LIN {X 0,Y 389.049,Z 504.507,A -85,B 0,C 180,E1 -11720.074,E2 -11720.074} C_VEL
LIN {X 0,Y 389.166,Z 500.329,A -85,B 0,C 180,E1 -11723.41,E2 -11723.41} C_VEL
LIN {X 0,Y 389.351,Z 496.924,A -85,B 0,C 180,E1 -11726.247,E2 -11726.247} C_VEL
LIN {X 0,Y 389.873,Z 499.181,A -85,B 0,C 180,E1 -11727.366,E2 -11727.366} C_VEL
LIN {X 0,Y 389.734,Z 506.684,A -85,B 0,C 180,E1 -11730.926,E2 -11730.926} C_VEL
LIN {X 0,Y 389.566,Z 513.106,A -85,B 0,C 180,E1 -11734.005,E2 -11734.005} C_VEL
LIN {X 0,Y 389.452,Z 518.341,A -85,B 0,C 180,E1 -11736.549,E2 -11736.549} C_VEL
LIN {X 0,Y 389.235,Z 525.161,A -85,B 0,C 180,E1 -11739.865,E2 -11739.865} C_VEL
LIN {X 0,Y 389.197,Z 528.183,A -85,B 0,C 180,E1 -11741.336,E2 -11741.336} C_VEL
LIN {X 0,Y 391.433,Z 539.991,A -85,B 0,C 180,E1 -11741.917,E2 -11741.917} C_VEL
LIN {X 0,Y 392.651,Z 549.622,A -85,B 0,C 180,E1 -11742.527,E2 -11742.527} C_VEL
LIN {X 0,Y 392.07,Z 559.282,A -85,B 0,C 180,E1 -11743.262,E2 -11743.262} C_VEL
LIN {X 0,Y 391.528,Z 567.985,A -85,B 0,C 180,E1 -11744.109,E2 -11744.109} C_VEL
LIN {X 0,Y 391.008,Z 575.053,A -85,B 0,C 180,E1 -11744.949,E2 -11744.949} C_VEL
LIN {X 0,Y 390.507,Z 581.055,A -85,B 0,C 180,E1 -11745.798,E2 -11745.798} C_VEL
LIN {X 0,Y 390.083,Z 586.933,A -85,B 0,C 180,E1 -11746.793,E2 -11746.793} C_VEL
LIN {X 0,Y 389.589,Z 593.354,A -85,B 0,C 180,E1 -11748.128,E2 -11748.128} C_VEL
LIN {X 0,Y 389.178,Z 599.487,A -85,B 0,C 180,E1 -11749.789,E2 -11749.789} C_VEL
LIN {X 0,Y 388.96,Z 602.788,A -85,B 0,C 180,E1 -11750.983,E2 -11750.983} C_VEL
LIN {X 0,Y 388.792,Z 605.13,A -85,B 0,C 180,E1 -11752.076,E2 -11752.076} C_VEL
LIN {X 0,Y 388.611,Z 607.077,A -85,B 0,C 180,E1 -11753.358,E2 -11753.358} C_VEL
LIN {X 0,Y 388.533,Z 608.221,A -85,B 0,C 180,E1 -11754.631,E2 -11754.631} C_VEL
LIN {X 0,Y 388.489,Z 608.513,A -85,B 0,C 180,E1 -11756.322,E2 -11756.322} C_VEL
LIN {X 0,Y 388.489,Z 608.255,A -85,B 0,C 180,E1 -11757.131,E2 -11757.131} C_VEL
LIN {X 0,Y 388.571,Z 607.186,A -85,B 0,C 180,E1 -11758.364,E2 -11758.364} C_VEL
LIN {X 0,Y 388.745,Z 605.399,A -85,B 0,C 180,E1 -11759.588,E2 -11759.588} C_VEL
LIN {X 0,Y 388.944,Z 601.354,A -85,B 0,C 180,E1 -11761.39,E2 -11761.39} C_VEL
LIN {X 0,Y 389.209,Z 597.195,A -85,B 0,C 180,E1 -11762.713,E2 -11762.713} C_VEL
LIN {X 0,Y 389.481,Z 593.091,A -85,B 0,C 180,E1 -11763.762,E2 -11763.762} C_VEL
LIN {X 0,Y 389.868,Z 587.471,A -85,B 0,C 180,E1 -11764.936,E2 -11764.936} C_VEL
LIN {X 0,Y 390.201,Z 582.47,A -85,B 0,C 180,E1 -11765.81,E2 -11765.81} C_VEL
LIN {X 0,Y 390.697,Z 575.482,A -85,B 0,C 180,E1 -11766.827,E2 -11766.827} C_VEL
LIN {X 0,Y 391.169,Z 568.265,A -85,B 0,C 180,E1 -11767.694,E2 -11767.694} C_VEL
LIN {X 0,Y 391.642,Z 559.908,A -85,B 0,C 180,E1 -11768.515,E2 -11768.515} C_VEL
LIN {X 0,Y 392.198,Z 550.305,A -85,B 0,C 180,E1 -11769.262,E2 -11769.262} C_VEL
LIN {X 0,Y 391.067,Z 540.77,A -85,B 0,C 180,E1 -11769.873,E2 -11769.873} C_VEL
LIN {X 0,Y 389.276,Z 529.916,A -85,B 0,C 180,E1 -11770.385,E2 -11770.385} C_VEL
LIN {X 0,Y 388.993,Z 528.206,A -85,B 0,C 180,E1 -11770.473,E2 -11770.473} C_VEL
LIN {X 0,Y 389.132,Z 520.919,A -85,B 0,C 180,E1 -11774.281,E2 -11774.281} C_VEL
LIN {X 0,Y 389.368,Z 513.777,A -85,B 0,C 180,E1 -11778.019,E2 -11778.019} C_VEL
LIN {X 0,Y 389.503,Z 506.789,A -85,B 0,C 180,E1 -11781.7,E2 -11781.7} C_VEL
LIN {X 0,Y 389.702,Z 499.725,A -85,B 0,C 180,E1 -11785.345,E2 -11785.345} C_VEL
LIN {X 0,Y 389.768,Z 496.75,A -85,B 0,C 180,E1 -11786.899,E2 -11786.899} C_VEL
LIN {X 0,Y 390.538,Z 496.652,A -85,B 0,C 180,E1 -11789.999,E2 -11789.999} C_VEL
LIN {X 0,Y 390.316,Z 496.677,A -85,B 0,C 180,E1 -11793.096,E2 -11793.096} C_VEL
LIN {X 0,Y 390.332,Z 496.678,A -85,B 0,C 180,E1 -11796.201,E2 -11796.201} C_VEL
LIN {X 0,Y 390.316,Z 496.68,A -85,B 0,C 180,E1 -11798.282,E2 -11798.282} C_VEL
LIN {X 0,Y 390.171,Z 496.698,A -85,B 0,C 180,E1 -11802.483,E2 -11802.483} C_VEL
LIN {X 0,Y 390.129,Z 496.7,A -85,B 0,C 180,E1 -11804.935,E2 -11804.935} C_VEL
LIN {X 0,Y 389.455,Z 496.787,A -85,B 0,C 180,E1 -11805.797,E2 -11805.797} C_VEL
LIN {X 0,Y 386.606,Z 497.139,A -85,B 0,C 180,E1 -11807.198,E2 -11807.198} C_VEL
LIN {X 0,Y 384.191,Z 497.444,A -85,B 0,C 180,E1 -11808.33,E2 -11808.33} C_VEL
LIN {X 0,Y 383.141,Z 497.57,A -85,B 0,C 180,E1 -11809.206,E2 -11809.206} C_VEL
LIN {X 0,Y 383.048,Z 497.581,A -85,B 0,C 180,E1 -11809.502,E2 -11809.502} C_VEL
LIN {X 0,Y 383.038,Z 497.583,A -85,B 0,C 180,E1 -11813.45,E2 -11813.45} C_VEL
LIN {X 0,Y 383.079,Z 497.582,A -85,B 0,C 180,E1 -11816.123,E2 -11816.123} C_VEL
LIN {X 0,Y 383.049,Z 497.585,A -85,B 0,C 180,E1 -11818.491,E2 -11818.491} C_VEL
LIN {X 0,Y 383.011,Z 497.591,A -85,B 0,C 180,E1 -11822.149,E2 -11822.149} C_VEL
LIN {X 0,Y 383.017,Z 497.587,A -85,B 0,C 180,E1 -11824.667,E2 -11824.667} C_VEL
LIN {X 0,Y 383.001,Z 497.591,A -85,B 0,C 180,E1 -11827.904,E2 -11827.904} C_VEL
LIN {X 0,Y 382.984,Z 497.59,A -85,B 0,C 180,E1 -11831.347,E2 -11831.347} C_VEL
LIN {X 0,Y 383.009,Z 497.59,A -85,B 0,C 180,E1 -11834.305,E2 -11834.305} C_VEL
LIN {X 0,Y 383.073,Z 497.578,A -85,B 0,C 180,E1 -11837.249,E2 -11837.249} C_VEL
LIN {X 0,Y 383.02,Z 497.588,A -85,B 0,C 180,E1 -11840.412,E2 -11840.412} C_VEL
LIN {X 0,Y 383.024,Z 497.589,A -85,B 0,C 180,E1 -11844.044,E2 -11844.044} C_VEL
LIN {X 0,Y 382.984,Z 497.592,A -85,B 0,C 180,E1 -11847.578,E2 -11847.578} C_VEL
LIN {X 0,Y 382.989,Z 497.592,A -85,B 0,C 180,E1 -11850.3,E2 -11850.3} C_VEL
LIN {X 0,Y 383.078,Z 497.582,A -85,B 0,C 180,E1 -11854.02,E2 -11854.02} C_VEL
LIN {X 0,Y 383.006,Z 497.588,A -85,B 0,C 180,E1 -11857.335,E2 -11857.335} C_VEL
LIN {X 0,Y 383.058,Z 497.58,A -85,B 0,C 180,E1 -11860.716,E2 -11860.716} C_VEL
LIN {X 0,Y 383.079,Z 497.582,A -85,B 0,C 180,E1 -11864.026,E2 -11864.026} C_VEL
LIN {X 0,Y 383.139,Z 497.571,A -85,B 0,C 180,E1 -11867.284,E2 -11867.284} C_VEL
LIN {X 0,Y 383.154,Z 497.569,A -85,B 0,C 180,E1 -11870.498,E2 -11870.498} C_VEL
LIN {X 0,Y 383.27,Z 497.554,A -85,B 0,C 180,E1 -11872.625,E2 -11872.625} C_VEL
LIN {X 0,Y 383.197,Z 497.563,A -85,B 0,C 180,E1 -11874.738,E2 -11874.738} C_VEL
LIN {X 0,Y 383.386,Z 497.544,A -85,B 0,C 180,E1 -11877.899,E2 -11877.899} C_VEL
LIN {X 0,Y 383.517,Z 497.527,A -85,B 0,C 180,E1 -11880,E2 -11880} C_VEL
LIN {X 0,Y 383.251,Z 497.558,A -85,B 0,C 180,E1 -11883.154,E2 -11883.154} C_VEL
LIN {X 0,Y 383.285,Z 497.553,A -85,B 0,C 180,E1 -11886.316,E2 -11886.316} C_VEL
LIN {X 0,Y 383.258,Z 497.556,A -85,B 0,C 180,E1 -11888.436,E2 -11888.436} C_VEL
LIN {X 0,Y 383.096,Z 497.58,A -85,B 0,C 180,E1 -11891.642,E2 -11891.642} C_VEL
LIN {X 0,Y 383.107,Z 497.575,A -85,B 0,C 180,E1 -11894.882,E2 -11894.882} C_VEL
LIN {X 0,Y 383.06,Z 497.581,A -85,B 0,C 180,E1 -11898.174,E2 -11898.174} C_VEL
LIN {X 0,Y 382.99,Z 497.593,A -85,B 0,C 180,E1 -11901.531,E2 -11901.531} C_VEL
LIN {X 0,Y 383.049,Z 497.582,A -85,B 0,C 180,E1 -11904.96,E2 -11904.96} C_VEL
LIN {X 0,Y 383.046,Z 497.582,A -85,B 0,C 180,E1 -11908.492,E2 -11908.492} C_VEL
LIN {X 0,Y 383.005,Z 497.587,A -85,B 0,C 180,E1 -11912.427,E2 -11912.427} C_VEL
LIN {X 0,Y 383.024,Z 497.587,A -85,B 0,C 180,E1 -11915.956,E2 -11915.956} C_VEL
LIN {X 0,Y 383.013,Z 497.59,A -85,B 0,C 180,E1 -11919.587,E2 -11919.587} C_VEL
LIN {X 0,Y 383.002,Z 497.588,A -85,B 0,C 180,E1 -11922.779,E2 -11922.779} C_VEL
LIN {X 0,Y 382.996,Z 497.592,A -85,B 0,C 180,E1 -11925.79,E2 -11925.79} C_VEL
LIN {X 0,Y 383.013,Z 497.587,A -85,B 0,C 180,E1 -11928.792,E2 -11928.792} C_VEL
LIN {X 0,Y 383.002,Z 497.59,A -85,B 0,C 180,E1 -11932.096,E2 -11932.096} C_VEL
LIN {X 0,Y 383.051,Z 497.676,A -85,B 0,C 180,E1 -11933.309,E2 -11933.309} C_VEL
LIN {X 0,Y 384.076,Z 503.252,A -85,B 0,C 180,E1 -11936.103,E2 -11936.103} C_VEL
LIN {X 0,Y 384.649,Z 507.173,A -85,B 0,C 180,E1 -11938.004,E2 -11938.004} C_VEL
LIN {X 0,Y 384.181,Z 513.651,A -85,B 0,C 180,E1 -11940.982,E2 -11940.982} C_VEL
LIN {X 0,Y 383.461,Z 521.478,A -85,B 0,C 180,E1 -11944.488,E2 -11944.488} C_VEL
LIN {X 0,Y 382.882,Z 529.232,A -85,B 0,C 180,E1 -11947.897,E2 -11947.897} C_VEL
LIN {X 0,Y 382.364,Z 538.246,A -85,B 0,C 180,E1 -11951.793,E2 -11951.793} C_VEL
LIN {X 0,Y 382.008,Z 546.977,A -85,B 0,C 180,E1 -11955.524,E2 -11955.524} C_VEL
LIN {X 0,Y 383.204,Z 558.101,A -85,B 0,C 180,E1 -11955.964,E2 -11955.964} C_VEL
LIN {X 0,Y 384.171,Z 569.277,A -85,B 0,C 180,E1 -11956.589,E2 -11956.589} C_VEL
LIN {X 0,Y 384.332,Z 577.789,A -85,B 0,C 180,E1 -11957.216,E2 -11957.216} C_VEL
LIN {X 0,Y 383.755,Z 587.394,A -85,B 0,C 180,E1 -11958.111,E2 -11958.111} C_VEL
LIN {X 0,Y 383.292,Z 595.307,A -85,B 0,C 180,E1 -11959.034,E2 -11959.034} C_VEL
LIN {X 0,Y 382.818,Z 601.82,A -85,B 0,C 180,E1 -11959.956,E2 -11959.956} C_VEL
LIN {X 0,Y 382.428,Z 607.997,A -85,B 0,C 180,E1 -11961.014,E2 -11961.014} C_VEL
LIN {X 0,Y 382.075,Z 614.282,A -85,B 0,C 180,E1 -11962.337,E2 -11962.337} C_VEL
LIN {X 0,Y 381.784,Z 619.534,A -85,B 0,C 180,E1 -11963.745,E2 -11963.745} C_VEL
LIN {X 0,Y 381.734,Z 623.67,A -85,B 0,C 180,E1 -11965.248,E2 -11965.248} C_VEL
LIN {X 0,Y 381.61,Z 626.719,A -85,B 0,C 180,E1 -11966.833,E2 -11966.833} C_VEL
LIN {X 0,Y 381.628,Z 628.092,A -85,B 0,C 180,E1 -11967.89,E2 -11967.89} C_VEL
LIN {X 0,Y 381.669,Z 628.965,A -85,B 0,C 180,E1 -11968.945,E2 -11968.945} C_VEL
LIN {X 0,Y 381.681,Z 629.274,A -85,B 0,C 180,E1 -11970.001,E2 -11970.001} C_VEL
LIN {X 0,Y 381.669,Z 629.017,A -85,B 0,C 180,E1 -11971.056,E2 -11971.056} C_VEL
LIN {X 0,Y 381.623,Z 628.273,A -85,B 0,C 180,E1 -11972.111,E2 -11972.111} C_VEL
LIN {X 0,Y 381.599,Z 627.035,A -85,B 0,C 180,E1 -11973.168,E2 -11973.168} C_VEL
LIN {X 0,Y 381.736,Z 624.119,A -85,B 0,C 180,E1 -11974.753,E2 -11974.753} C_VEL
LIN {X 0,Y 381.751,Z 621.238,A -85,B 0,C 180,E1 -11975.884,E2 -11975.884} C_VEL
LIN {X 0,Y 382.042,Z 616.321,A -85,B 0,C 180,E1 -11977.399,E2 -11977.399} C_VEL
LIN {X 0,Y 382.397,Z 611.016,A -85,B 0,C 180,E1 -11978.722,E2 -11978.722} C_VEL
LIN {X 0,Y 382.939,Z 604.445,A -85,B 0,C 180,E1 -11980.041,E2 -11980.041} C_VEL
LIN {X 0,Y 383.679,Z 596.352,A -85,B 0,C 180,E1 -11981.357,E2 -11981.357} C_VEL
LIN {X 0,Y 384.433,Z 587.126,A -85,B 0,C 180,E1 -11982.539,E2 -11982.539} C_VEL
LIN {X 0,Y 385.246,Z 578.244,A -85,B 0,C 180,E1 -11983.451,E2 -11983.451} C_VEL
LIN {X 0,Y 385.214,Z 569.496,A -85,B 0,C 180,E1 -11984.227,E2 -11984.227} C_VEL
LIN {X 0,Y 384.556,Z 559.789,A -85,B 0,C 180,E1 -11984.96,E2 -11984.96} C_VEL
LIN {X 0,Y 382.593,Z 547.8,A -85,B 0,C 180,E1 -11985.73,E2 -11985.73} C_VEL
LIN {X 0,Y 382.063,Z 545.124,A -85,B 0,C 180,E1 -11985.881,E2 -11985.881} C_VEL
LIN {X 0,Y 382.441,Z 537.733,A -85,B 0,C 180,E1 -11989.317,E2 -11989.317} C_VEL
LIN {X 0,Y 382.895,Z 530.876,A -85,B 0,C 180,E1 -11992.672,E2 -11992.672} C_VEL
LIN {X 0,Y 383.459,Z 525.387,A -85,B 0,C 180,E1 -11995.513,E2 -11995.513} C_VEL
LIN {X 0,Y 384.131,Z 519.884,A -85,B 0,C 180,E1 -11998.574,E2 -11998.574} C_VEL
LIN {X 0,Y 384.904,Z 514.395,A -85,B 0,C 180,E1 -12001.973,E2 -12001.973} C_VEL
LIN {X 0,Y 385.185,Z 510.943,A -85,B 0,C 180,E1 -12004.446,E2 -12004.446} C_VEL
LIN {X 0,Y 384.805,Z 507.931,A -85,B 0,C 180,E1 -12007.064,E2 -12007.064} C_VEL
LIN {X 0,Y 384.399,Z 505.368,A -85,B 0,C 180,E1 -12009.835,E2 -12009.835} C_VEL
LIN {X 0,Y 384.03,Z 503.279,A -85,B 0,C 180,E1 -12012.944,E2 -12012.944} C_VEL
LIN {X 0,Y 383.811,Z 502.03,A -85,B 0,C 180,E1 -12015.907,E2 -12015.907} C_VEL
LIN {X 0,Y 383.693,Z 501.503,A -85,B 0,C 180,E1 -12018.746,E2 -12018.746} C_VEL
LIN {X 0,Y 383.687,Z 501.616,A -85,B 0,C 180,E1 -12021.966,E2 -12021.966} C_VEL
LIN {X 0,Y 383.733,Z 502.06,A -85,B 0,C 180,E1 -12024.121,E2 -12024.121} C_VEL
LIN {X 0,Y 383.785,Z 503.255,A -85,B 0,C 180,E1 -12027.392,E2 -12027.392} C_VEL
LIN {X 0,Y 383.465,Z 504.845,A -85,B 0,C 180,E1 -12030.34,E2 -12030.34} C_VEL
LIN {X 0,Y 383.059,Z 507.299,A -85,B 0,C 180,E1 -12034.029,E2 -12034.029} C_VEL
LIN {X 0,Y 382.756,Z 509.832,A -85,B 0,C 180,E1 -12037.32,E2 -12037.32} C_VEL
LIN {X 0,Y 382.535,Z 512.699,A -85,B 0,C 180,E1 -12040.689,E2 -12040.689} C_VEL
LIN {X 0,Y 382.316,Z 516.009,A -85,B 0,C 180,E1 -12044.276,E2 -12044.276} C_VEL
LIN {X 0,Y 385.469,Z 526.823,A -85,B 0,C 180,E1 -12045.088,E2 -12045.088} C_VEL
LIN {X 0,Y 386.98,Z 535.241,A -85,B 0,C 180,E1 -12045.792,E2 -12045.792} C_VEL
LIN {X 0,Y 386.311,Z 544.52,A -85,B 0,C 180,E1 -12046.588,E2 -12046.588} C_VEL
LIN {X 0,Y 385.581,Z 553.105,A -85,B 0,C 180,E1 -12047.5,E2 -12047.5} C_VEL
LIN {X 0,Y 384.783,Z 562.092,A -85,B 0,C 180,E1 -12048.677,E2 -12048.677} C_VEL
LIN {X 0,Y 383.992,Z 569.911,A -85,B 0,C 180,E1 -12049.987,E2 -12049.987} C_VEL
LIN {X 0,Y 383.385,Z 576.206,A -85,B 0,C 180,E1 -12051.302,E2 -12051.302} C_VEL
LIN {X 0,Y 382.925,Z 581.247,A -85,B 0,C 180,E1 -12052.619,E2 -12052.619} C_VEL
LIN {X 0,Y 382.358,Z 585.933,A -85,B 0,C 180,E1 -12054.198,E2 -12054.198} C_VEL
LIN {X 0,Y 382.23,Z 589.116,A -85,B 0,C 180,E1 -12055.782,E2 -12055.782} C_VEL
LIN {X 0,Y 381.996,Z 590.639,A -85,B 0,C 180,E1 -12056.836,E2 -12056.836} C_VEL
LIN {X 0,Y 381.838,Z 591.561,A -85,B 0,C 180,E1 -12057.89,E2 -12057.89} C_VEL
LIN {X 0,Y 381.72,Z 591.956,A -85,B 0,C 180,E1 -12058.945,E2 -12058.945} C_VEL
LIN {X 0,Y 381.684,Z 591.867,A -85,B 0,C 180,E1 -12060,E2 -12060} C_VEL
LIN {X 0,Y 381.708,Z 591.289,A -85,B 0,C 180,E1 -12061.055,E2 -12061.055} C_VEL
LIN {X 0,Y 381.79,Z 590.191,A -85,B 0,C 180,E1 -12062.11,E2 -12062.11} C_VEL
LIN {X 0,Y 381.823,Z 587.432,A -85,B 0,C 180,E1 -12063.694,E2 -12063.694} C_VEL
LIN {X 0,Y 381.942,Z 584.941,A -85,B 0,C 180,E1 -12064.75,E2 -12064.75} C_VEL
LIN {X 0,Y 382.161,Z 579.878,A -85,B 0,C 180,E1 -12066.335,E2 -12066.335} C_VEL
LIN {X 0,Y 382.451,Z 575.661,A -85,B 0,C 180,E1 -12067.391,E2 -12067.391} C_VEL
LIN {X 0,Y 382.636,Z 570.597,A -85,B 0,C 180,E1 -12068.45,E2 -12068.45} C_VEL
LIN {X 0,Y 383.015,Z 564.521,A -85,B 0,C 180,E1 -12069.506,E2 -12069.506} C_VEL
LIN {X 0,Y 383.538,Z 556.171,A -85,B 0,C 180,E1 -12070.692,E2 -12070.692} C_VEL
LIN {X 0,Y 384.064,Z 547.02,A -85,B 0,C 180,E1 -12071.746,E2 -12071.746} C_VEL
LIN {X 0,Y 384.611,Z 536.714,A -85,B 0,C 180,E1 -12072.667,E2 -12072.667} C_VEL
LIN {X 0,Y 384.733,Z 530.686,A -85,B 0,C 180,E1 -12073.117,E2 -12073.117} C_VEL
LIN {X 0,Y 382.871,Z 519.137,A -85,B 0,C 180,E1 -12073.823,E2 -12073.823} C_VEL
LIN {X 0,Y 381.887,Z 512.68,A -85,B 0,C 180,E1 -12074.148,E2 -12074.148} C_VEL
LIN {X 0,Y 381.92,Z 508.837,A -85,B 0,C 180,E1 -12077.123,E2 -12077.123} C_VEL
LIN {X 0,Y 381.983,Z 504.619,A -85,B 0,C 180,E1 -12080.461,E2 -12080.461} C_VEL
LIN {X 0,Y 382.102,Z 500.414,A -85,B 0,C 180,E1 -12083.869,E2 -12083.869} C_VEL
LIN {X 0,Y 382.27,Z 497.752,A -85,B 0,C 180,E1 -12086.112,E2 -12086.112} C_VEL
LIN {X 0,Y 382.862,Z 500.164,A -85,B 0,C 180,E1 -12087.317,E2 -12087.317} C_VEL
LIN {X 0,Y 382.73,Z 506.454,A -85,B 0,C 180,E1 -12090.338,E2 -12090.338} C_VEL
LIN {X 0,Y 382.597,Z 512.872,A -85,B 0,C 180,E1 -12093.441,E2 -12093.441} C_VEL
LIN {X 0,Y 382.4,Z 519.478,A -85,B 0,C 180,E1 -12096.677,E2 -12096.677} C_VEL
LIN {X 0,Y 382.185,Z 526.372,A -85,B 0,C 180,E1 -12100.062,E2 -12100.062} C_VEL
LIN {X 0,Y 382.151,Z 528.35,A -85,B 0,C 180,E1 -12101.037,E2 -12101.037} C_VEL
LIN {X 0,Y 384.343,Z 539.751,A -85,B 0,C 180,E1 -12101.606,E2 -12101.606} C_VEL
LIN {X 0,Y 385.754,Z 550.364,A -85,B 0,C 180,E1 -12102.296,E2 -12102.296} C_VEL
LIN {X 0,Y 385.116,Z 560.662,A -85,B 0,C 180,E1 -12103.116,E2 -12103.116} C_VEL
LIN {X 0,Y 384.561,Z 569.215,A -85,B 0,C 180,E1 -12103.985,E2 -12103.985} C_VEL
LIN {X 0,Y 383.934,Z 576.895,A -85,B 0,C 180,E1 -12104.944,E2 -12104.944} C_VEL
LIN {X 0,Y 383.288,Z 584.991,A -85,B 0,C 180,E1 -12106.196,E2 -12106.196} C_VEL
LIN {X 0,Y 382.687,Z 591.911,A -85,B 0,C 180,E1 -12107.582,E2 -12107.582} C_VEL
LIN {X 0,Y 382.305,Z 597.184,A -85,B 0,C 180,E1 -12108.913,E2 -12108.913} C_VEL
LIN {X 0,Y 382.055,Z 600.427,A -85,B 0,C 180,E1 -12109.921,E2 -12109.921} C_VEL
LIN {X 0,Y 381.823,Z 603.802,A -85,B 0,C 180,E1 -12111.257,E2 -12111.257} C_VEL
LIN {X 0,Y 381.653,Z 606.232,A -85,B 0,C 180,E1 -12112.577,E2 -12112.577} C_VEL
LIN {X 0,Y 381.468,Z 608.058,A -85,B 0,C 180,E1 -12114.158,E2 -12114.158} C_VEL
LIN {X 0,Y 381.394,Z 608.789,A -85,B 0,C 180,E1 -12116.019,E2 -12116.019} C_VEL
LIN {X 0,Y 381.443,Z 607.778,A -85,B 0,C 180,E1 -12117.945,E2 -12117.945} C_VEL
LIN {X 0,Y 381.561,Z 606.623,A -85,B 0,C 180,E1 -12118.953,E2 -12118.953} C_VEL
LIN {X 0,Y 381.692,Z 604.535,A -85,B 0,C 180,E1 -12120.188,E2 -12120.188} C_VEL
LIN {X 0,Y 381.985,Z 599.971,A -85,B 0,C 180,E1 -12122.023,E2 -12122.023} C_VEL
LIN {X 0,Y 382.355,Z 594.798,A -85,B 0,C 180,E1 -12123.529,E2 -12123.529} C_VEL
LIN {X 0,Y 382.779,Z 589.025,A -85,B 0,C 180,E1 -12124.816,E2 -12124.816} C_VEL
LIN {X 0,Y 383.162,Z 583.003,A -85,B 0,C 180,E1 -12125.913,E2 -12125.913} C_VEL
LIN {X 0,Y 383.69,Z 576.046,A -85,B 0,C 180,E1 -12126.953,E2 -12126.953} C_VEL
LIN {X 0,Y 384.168,Z 568.93,A -85,B 0,C 180,E1 -12127.832,E2 -12127.832} C_VEL
LIN {X 0,Y 384.594,Z 561.818,A -85,B 0,C 180,E1 -12128.563,E2 -12128.563} C_VEL
LIN {X 0,Y 385.161,Z 553.061,A -85,B 0,C 180,E1 -12129.289,E2 -12129.289} C_VEL
LIN {X 0,Y 385.144,Z 548.708,A -85,B 0,C 180,E1 -12129.608,E2 -12129.608} C_VEL
LIN {X 0,Y 383.53,Z 537.804,A -85,B 0,C 180,E1 -12130.272,E2 -12130.272} C_VEL
LIN {X 0,Y 381.934,Z 528.331,A -85,B 0,C 180,E1 -12130.726,E2 -12130.726} C_VEL
LIN {X 0,Y 382.066,Z 521.137,A -85,B 0,C 180,E1 -12134.53,E2 -12134.53} C_VEL
LIN {X 0,Y 382.332,Z 513.945,A -85,B 0,C 180,E1 -12138.334,E2 -12138.334} C_VEL
LIN {X 0,Y 382.444,Z 507.836,A -85,B 0,C 180,E1 -12141.546,E2 -12141.546} C_VEL
LIN {X 0,Y 382.671,Z 500.777,A -85,B 0,C 180,E1 -12145.259,E2 -12145.259} C_VEL
LIN {X 0,Y 382.743,Z 497.625,A -85,B 0,C 180,E1 -12146.973,E2 -12146.973} C_VEL
LIN {X 0,Y 383.485,Z 497.53,A -85,B 0,C 180,E1 -12149.999,E2 -12149.999} C_VEL
LIN {X 0,Y 383.252,Z 497.556,A -85,B 0,C 180,E1 -12153.153,E2 -12153.153} C_VEL
LIN {X 0,Y 383.289,Z 497.556,A -85,B 0,C 180,E1 -12156.316,E2 -12156.316} C_VEL
LIN {X 0,Y 383.261,Z 497.559,A -85,B 0,C 180,E1 -12158.435,E2 -12158.435} C_VEL
LIN {X 0,Y 383.098,Z 497.577,A -85,B 0,C 180,E1 -12161.642,E2 -12161.642} C_VEL
LIN {X 0,Y 383.108,Z 497.574,A -85,B 0,C 180,E1 -12164.921,E2 -12164.921} C_VEL
LIN {X 0,Y 383.09,Z 497.581,A -85,B 0,C 180,E1 -12168.172,E2 -12168.172} C_VEL
LIN {X 0,Y 383.048,Z 497.581,A -85,B 0,C 180,E1 -12169.502,E2 -12169.502} C_VEL
LIN {X 0,Y 382.358,Z 497.672,A -85,B 0,C 180,E1 -12170.379,E2 -12170.379} C_VEL
LIN {X 0,Y 379.491,Z 498.026,A -85,B 0,C 180,E1 -12171.805,E2 -12171.805} C_VEL
LIN {X 0,Y 377.085,Z 498.325,A -85,B 0,C 180,E1 -12172.957,E2 -12172.957} C_VEL
LIN {X 0,Y 376.067,Z 498.454,A -85,B 0,C 180,E1 -12173.848,E2 -12173.848} C_VEL
LIN {X 0,Y 375.99,Z 498.464,A -85,B 0,C 180,E1 -12174.15,E2 -12174.15} C_VEL
LIN {X 0,Y 376.019,Z 498.459,A -85,B 0,C 180,E1 -12176.651,E2 -12176.651} C_VEL
LIN {X 0,Y 375.976,Z 498.462,A -85,B 0,C 180,E1 -12179.078,E2 -12179.078} C_VEL
LIN {X 0,Y 375.951,Z 498.466,A -85,B 0,C 180,E1 -12182.828,E2 -12182.828} C_VEL
LIN {X 0,Y 375.957,Z 498.465,A -85,B 0,C 180,E1 -12185.415,E2 -12185.415} C_VEL
LIN {X 0,Y 375.975,Z 498.467,A -85,B 0,C 180,E1 -12188.27,E2 -12188.27} C_VEL
LIN {X 0,Y 375.934,Z 498.469,A -85,B 0,C 180,E1 -12191.6,E2 -12191.6} C_VEL
LIN {X 0,Y 375.98,Z 498.462,A -85,B 0,C 180,E1 -12195.26,E2 -12195.26} C_VEL
LIN {X 0,Y 375.988,Z 498.464,A -85,B 0,C 180,E1 -12198.389,E2 -12198.389} C_VEL
LIN {X 0,Y 375.966,Z 498.468,A -85,B 0,C 180,E1 -12201.912,E2 -12201.912} C_VEL
LIN {X 0,Y 375.977,Z 498.463,A -85,B 0,C 180,E1 -12205.332,E2 -12205.332} C_VEL
LIN {X 0,Y 375.955,Z 498.467,A -85,B 0,C 180,E1 -12208.438,E2 -12208.438} C_VEL
LIN {X 0,Y 375.981,Z 498.466,A -85,B 0,C 180,E1 -12212.14,E2 -12212.14} C_VEL
LIN {X 0,Y 376.004,Z 498.46,A -85,B 0,C 180,E1 -12214.539,E2 -12214.539} C_VEL
LIN {X 0,Y 375.961,Z 498.468,A -85,B 0,C 180,E1 -12218.045,E2 -12218.045} C_VEL
LIN {X 0,Y 376.021,Z 498.459,A -85,B 0,C 180,E1 -12221.474,E2 -12221.474} C_VEL
LIN {X 0,Y 376.057,Z 498.452,A -85,B 0,C 180,E1 -12224.832,E2 -12224.832} C_VEL
LIN {X 0,Y 376.056,Z 498.456,A -85,B 0,C 180,E1 -12228.137,E2 -12228.137} C_VEL
LIN {X 0,Y 376.255,Z 498.433,A -85,B 0,C 180,E1 -12231.877,E2 -12231.877} C_VEL
LIN {X 0,Y 376.17,Z 498.438,A -85,B 0,C 180,E1 -12234.64,E2 -12234.64} C_VEL
LIN {X 0,Y 376.352,Z 498.42,A -85,B 0,C 180,E1 -12237.86,E2 -12237.86} C_VEL
LIN {X 0,Y 376.486,Z 498.403,A -85,B 0,C 180,E1 -12240,E2 -12240} C_VEL
LIN {X 0,Y 376.189,Z 498.437,A -85,B 0,C 180,E1 -12243.213,E2 -12243.213} C_VEL
LIN {X 0,Y 376.244,Z 498.429,A -85,B 0,C 180,E1 -12246.435,E2 -12246.435} C_VEL
LIN {X 0,Y 376.203,Z 498.434,A -85,B 0,C 180,E1 -12248.595,E2 -12248.595} C_VEL
LIN {X 0,Y 376.048,Z 498.458,A -85,B 0,C 180,E1 -12251.863,E2 -12251.863} C_VEL
LIN {X 0,Y 376.055,Z 498.454,A -85,B 0,C 180,E1 -12255.167,E2 -12255.167} C_VEL
LIN {X 0,Y 376.006,Z 498.458,A -85,B 0,C 180,E1 -12258.527,E2 -12258.527} C_VEL
LIN {X 0,Y 375.96,Z 498.468,A -85,B 0,C 180,E1 -12261.954,E2 -12261.954} C_VEL
LIN {X 0,Y 376.004,Z 498.464,A -85,B 0,C 180,E1 -12265.461,E2 -12265.461} C_VEL
LIN {X 0,Y 375.974,Z 498.464,A -85,B 0,C 180,E1 -12269.079,E2 -12269.079} C_VEL
LIN {X 0,Y 375.955,Z 498.465,A -85,B 0,C 180,E1 -12272.828,E2 -12272.828} C_VEL
LIN {X 0,Y 375.955,Z 498.469,A -85,B 0,C 180,E1 -12275.416,E2 -12275.416} C_VEL
LIN {X 0,Y 375.973,Z 498.463,A -85,B 0,C 180,E1 -12278.271,E2 -12278.271} C_VEL
LIN {X 0,Y 375.932,Z 498.472,A -85,B 0,C 180,E1 -12281.601,E2 -12281.601} C_VEL
LIN {X 0,Y 375.951,Z 498.469,A -85,B 0,C 180,E1 -12285.265,E2 -12285.265} C_VEL
LIN {X 0,Y 375.979,Z 498.465,A -85,B 0,C 180,E1 -12289.139,E2 -12289.139} C_VEL
LIN {X 0,Y 376.03,Z 498.59,A -85,B 0,C 180,E1 -12293.185,E2 -12293.185} C_VEL
LIN {X 0,Y 377.019,Z 504.098,A -85,B 0,C 180,E1 -12295.998,E2 -12295.998} C_VEL
LIN {X 0,Y 377.631,Z 508.075,A -85,B 0,C 180,E1 -12297.968,E2 -12297.968} C_VEL
LIN {X 0,Y 377.085,Z 514.89,A -85,B 0,C 180,E1 -12301.16,E2 -12301.16} C_VEL
LIN {X 0,Y 376.359,Z 522.349,A -85,B 0,C 180,E1 -12304.565,E2 -12304.565} C_VEL
LIN {X 0,Y 375.767,Z 530.072,A -85,B 0,C 180,E1 -12308.034,E2 -12308.034} C_VEL
LIN {X 0,Y 375.253,Z 539.055,A -85,B 0,C 180,E1 -12312,E2 -12312} C_VEL
LIN {X 0,Y 374.905,Z 546.542,A -85,B 0,C 180,E1 -12315.272,E2 -12315.272} C_VEL
LIN {X 0,Y 375.987,Z 556.294,A -85,B 0,C 180,E1 -12315.644,E2 -12315.644} C_VEL
LIN {X 0,Y 376.795,Z 565.256,A -85,B 0,C 180,E1 -12316.121,E2 -12316.121} C_VEL
LIN {X 0,Y 377.407,Z 573.354,A -85,B 0,C 180,E1 -12316.677,E2 -12316.677} C_VEL
LIN {X 0,Y 377.212,Z 580.052,A -85,B 0,C 180,E1 -12317.218,E2 -12317.218} C_VEL
LIN {X 0,Y 376.716,Z 588.219,A -85,B 0,C 180,E1 -12318.022,E2 -12318.022} C_VEL
LIN {X 0,Y 376.215,Z 595.958,A -85,B 0,C 180,E1 -12318.962,E2 -12318.962} C_VEL
LIN {X 0,Y 375.683,Z 603.181,A -85,B 0,C 180,E1 -12320.036,E2 -12320.036} C_VEL
LIN {X 0,Y 375.223,Z 610.455,A -85,B 0,C 180,E1 -12321.383,E2 -12321.383} C_VEL
LIN {X 0,Y 374.979,Z 615.13,A -85,B 0,C 180,E1 -12322.462,E2 -12322.462} C_VEL
LIN {X 0,Y 374.677,Z 619.781,A -85,B 0,C 180,E1 -12323.797,E2 -12323.797} C_VEL
LIN {X 0,Y 374.645,Z 623.43,A -85,B 0,C 180,E1 -12325.158,E2 -12325.158} C_VEL
LIN {X 0,Y 374.522,Z 626.494,A -85,B 0,C 180,E1 -12326.773,E2 -12326.773} C_VEL
LIN {X 0,Y 374.526,Z 627.881,A -85,B 0,C 180,E1 -12327.85,E2 -12327.85} C_VEL
LIN {X 0,Y 374.569,Z 628.765,A -85,B 0,C 180,E1 -12328.925,E2 -12328.925} C_VEL
LIN {X 0,Y 374.612,Z 629.078,A -85,B 0,C 180,E1 -12330.001,E2 -12330.001} C_VEL
LIN {X 0,Y 374.569,Z 628.831,A -85,B 0,C 180,E1 -12331.076,E2 -12331.076} C_VEL
LIN {X 0,Y 374.521,Z 628.101,A -85,B 0,C 180,E1 -12332.151,E2 -12332.151} C_VEL
LIN {X 0,Y 374.512,Z 626.876,A -85,B 0,C 180,E1 -12333.228,E2 -12333.228} C_VEL
LIN {X 0,Y 374.648,Z 623.972,A -85,B 0,C 180,E1 -12334.843,E2 -12334.843} C_VEL
LIN {X 0,Y 374.76,Z 620.187,A -85,B 0,C 180,E1 -12336.318,E2 -12336.318} C_VEL
LIN {X 0,Y 375.111,Z 614.352,A -85,B 0,C 180,E1 -12338.078,E2 -12338.078} C_VEL
LIN {X 0,Y 375.575,Z 608.694,A -85,B 0,C 180,E1 -12339.424,E2 -12339.424} C_VEL
LIN {X 0,Y 376.253,Z 601.713,A -85,B 0,C 180,E1 -12340.766,E2 -12340.766} C_VEL
LIN {X 0,Y 377.146,Z 592.885,A -85,B 0,C 180,E1 -12342.102,E2 -12342.102} C_VEL
LIN {X 0,Y 377.795,Z 585.429,A -85,B 0,C 180,E1 -12343.036,E2 -12343.036} C_VEL
LIN {X 0,Y 378.525,Z 577.81,A -85,B 0,C 180,E1 -12343.831,E2 -12343.831} C_VEL
LIN {X 0,Y 378.406,Z 568.817,A -85,B 0,C 180,E1 -12344.652,E2 -12344.652} C_VEL
LIN {X 0,Y 377.711,Z 559.508,A -85,B 0,C 180,E1 -12345.376,E2 -12345.376} C_VEL
LIN {X 0,Y 375.376,Z 546.638,A -85,B 0,C 180,E1 -12346.25,E2 -12346.25} C_VEL
LIN {X 0,Y 375.047,Z 544.656,A -85,B 0,C 180,E1 -12346.378,E2 -12346.378} C_VEL
LIN {X 0,Y 375.536,Z 536.733,A -85,B 0,C 180,E1 -12350.186,E2 -12350.186} C_VEL
LIN {X 0,Y 376.189,Z 528.767,A -85,B 0,C 180,E1 -12354.269,E2 -12354.269} C_VEL
LIN {X 0,Y 376.902,Z 522.441,A -85,B 0,C 180,E1 -12357.786,E2 -12357.786} C_VEL
LIN {X 0,Y 377.729,Z 516.997,A -85,B 0,C 180,E1 -12361.144,E2 -12361.144} C_VEL
LIN {X 0,Y 378.164,Z 513.947,A -85,B 0,C 180,E1 -12363.248,E2 -12363.248} C_VEL
LIN {X 0,Y 378.176,Z 511.502,A -85,B 0,C 180,E1 -12365.177,E2 -12365.177} C_VEL
LIN {X 0,Y 377.657,Z 507.988,A -85,B 0,C 180,E1 -12368.593,E2 -12368.593} C_VEL
LIN {X 0,Y 377.209,Z 505.35,A -85,B 0,C 180,E1 -12372.125,E2 -12372.125} C_VEL
LIN {X 0,Y 376.937,Z 503.898,A -85,B 0,C 180,E1 -12375.115,E2 -12375.115} C_VEL
LIN {X 0,Y 376.758,Z 503.14,A -85,B 0,C 180,E1 -12378.259,E2 -12378.259} C_VEL
LIN {X 0,Y 376.755,Z 503.083,A -85,B 0,C 180,E1 -12381.58,E2 -12381.58} C_VEL
LIN {X 0,Y 376.785,Z 503.676,A -85,B 0,C 180,E1 -12384.674,E2 -12384.674} C_VEL
LIN {X 0,Y 376.818,Z 504.586,A -85,B 0,C 180,E1 -12387.257,E2 -12387.257} C_VEL
LIN {X 0,Y 376.551,Z 505.815,A -85,B 0,C 180,E1 -12389.74,E2 -12389.74} C_VEL
LIN {X 0,Y 376.249,Z 507.263,A -85,B 0,C 180,E1 -12392.162,E2 -12392.162} C_VEL
LIN {X 0,Y 375.993,Z 508.868,A -85,B 0,C 180,E1 -12394.538,E2 -12394.538} C_VEL
LIN {X 0,Y 375.691,Z 511.515,A -85,B 0,C 180,E1 -12398.029,E2 -12398.029} C_VEL
LIN {X 0,Y 375.454,Z 514.394,A -85,B 0,C 180,E1 -12401.445,E2 -12401.445} C_VEL
LIN {X 0,Y 375.296,Z 516.501,A -85,B 0,C 180,E1 -12403.782,E2 -12403.782} C_VEL
LIN {X 0,Y 378.338,Z 526.479,A -85,B 0,C 180,E1 -12404.579,E2 -12404.579} C_VEL
LIN {X 0,Y 380.327,Z 536.349,A -85,B 0,C 180,E1 -12405.458,E2 -12405.458} C_VEL
LIN {X 0,Y 379.665,Z 544.928,A -85,B 0,C 180,E1 -12406.212,E2 -12406.212} C_VEL
LIN {X 0,Y 379.009,Z 552.369,A -85,B 0,C 180,E1 -12407.007,E2 -12407.007} C_VEL
LIN {X 0,Y 378.318,Z 559.619,A -85,B 0,C 180,E1 -12407.937,E2 -12407.937} C_VEL
LIN {X 0,Y 377.416,Z 568.132,A -85,B 0,C 180,E1 -12409.268,E2 -12409.268} C_VEL
LIN {X 0,Y 376.693,Z 574.803,A -85,B 0,C 180,E1 -12410.605,E2 -12410.605} C_VEL
LIN {X 0,Y 376.099,Z 580.54,A -85,B 0,C 180,E1 -12412.052,E2 -12412.052} C_VEL
LIN {X 0,Y 375.422,Z 585.187,A -85,B 0,C 180,E1 -12413.551,E2 -12413.551} C_VEL
LIN {X 0,Y 375.288,Z 587.704,A -85,B 0,C 180,E1 -12414.627,E2 -12414.627} C_VEL
LIN {X 0,Y 375.193,Z 589.672,A -85,B 0,C 180,E1 -12415.703,E2 -12415.703} C_VEL
LIN {X 0,Y 374.948,Z 591.139,A -85,B 0,C 180,E1 -12416.777,E2 -12416.777} C_VEL
LIN {X 0,Y 374.778,Z 592.032,A -85,B 0,C 180,E1 -12417.851,E2 -12417.851} C_VEL
LIN {X 0,Y 374.654,Z 592.356,A -85,B 0,C 180,E1 -12418.925,E2 -12418.925} C_VEL
LIN {X 0,Y 374.616,Z 592.195,A -85,B 0,C 180,E1 -12420,E2 -12420} C_VEL
LIN {X 0,Y 374.642,Z 591.552,A -85,B 0,C 180,E1 -12421.075,E2 -12421.075} C_VEL
LIN {X 0,Y 374.694,Z 590.412,A -85,B 0,C 180,E1 -12422.15,E2 -12422.15} C_VEL
LIN {X 0,Y 374.736,Z 587.553,A -85,B 0,C 180,E1 -12423.764,E2 -12423.764} C_VEL
LIN {X 0,Y 374.922,Z 583.405,A -85,B 0,C 180,E1 -12425.378,E2 -12425.378} C_VEL
LIN {X 0,Y 375.101,Z 579.83,A -85,B 0,C 180,E1 -12426.455,E2 -12426.455} C_VEL
LIN {X 0,Y 375.427,Z 574.315,A -85,B 0,C 180,E1 -12427.8,E2 -12427.8} C_VEL
LIN {X 0,Y 375.784,Z 567.462,A -85,B 0,C 180,E1 -12429.147,E2 -12429.147} C_VEL
LIN {X 0,Y 376.322,Z 558.721,A -85,B 0,C 180,E1 -12430.491,E2 -12430.491} C_VEL
LIN {X 0,Y 376.807,Z 551.197,A -85,B 0,C 180,E1 -12431.43,E2 -12431.43} C_VEL
LIN {X 0,Y 377.226,Z 543.433,A -85,B 0,C 180,E1 -12432.235,E2 -12432.235} C_VEL
LIN {X 0,Y 377.695,Z 534.591,A -85,B 0,C 180,E1 -12432.982,E2 -12432.982} C_VEL
LIN {X 0,Y 377.552,Z 530.344,A -85,B 0,C 180,E1 -12433.305,E2 -12433.305} C_VEL
LIN {X 0,Y 375.743,Z 519.206,A -85,B 0,C 180,E1 -12433.992,E2 -12433.992} C_VEL
LIN {X 0,Y 374.792,Z 512.984,A -85,B 0,C 180,E1 -12434.317,E2 -12434.317} C_VEL
LIN {X 0,Y 374.849,Z 508.982,A -85,B 0,C 180,E1 -12437.457,E2 -12437.457} C_VEL
LIN {X 0,Y 374.912,Z 504.721,A -85,B 0,C 180,E1 -12440.865,E2 -12440.865} C_VEL
LIN {X 0,Y 375.058,Z 500.486,A -85,B 0,C 180,E1 -12444.346,E2 -12444.346} C_VEL
LIN {X 0,Y 375.217,Z 498.592,A -85,B 0,C 180,E1 -12445.964,E2 -12445.964} C_VEL
LIN {X 0,Y 375.848,Z 501.177,A -85,B 0,C 180,E1 -12447.266,E2 -12447.266} C_VEL
LIN {X 0,Y 375.69,Z 508.05,A -85,B 0,C 180,E1 -12450.624,E2 -12450.624} C_VEL
LIN {X 0,Y 375.477,Z 515.276,A -85,B 0,C 180,E1 -12454.162,E2 -12454.162} C_VEL
LIN {X 0,Y 375.306,Z 521.998,A -85,B 0,C 180,E1 -12457.469,E2 -12457.469} C_VEL
LIN {X 0,Y 375.069,Z 528.49,A -85,B 0,C 180,E1 -12460.708,E2 -12460.708} C_VEL
LIN {X 0,Y 377.511,Z 541.051,A -85,B 0,C 180,E1 -12461.367,E2 -12461.367} C_VEL
LIN {X 0,Y 378.883,Z 551.614,A -85,B 0,C 180,E1 -12462.1,E2 -12462.1} C_VEL
LIN {X 0,Y 378.285,Z 560.173,A -85,B 0,C 180,E1 -12462.789,E2 -12462.789} C_VEL
LIN {X 0,Y 377.732,Z 568.084,A -85,B 0,C 180,E1 -12463.585,E2 -12463.585} C_VEL
LIN {X 0,Y 377.099,Z 575.756,A -85,B 0,C 180,E1 -12464.531,E2 -12464.531} C_VEL
LIN {X 0,Y 376.398,Z 583.747,A -85,B 0,C 180,E1 -12465.744,E2 -12465.744} C_VEL
LIN {X 0,Y 375.758,Z 591.402,A -85,B 0,C 180,E1 -12467.232,E2 -12467.232} C_VEL
LIN {X 0,Y 375.353,Z 596.5,A -85,B 0,C 180,E1 -12468.5,E2 -12468.5} C_VEL
LIN {X 0,Y 374.909,Z 601.845,A -85,B 0,C 180,E1 -12470.227,E2 -12470.227} C_VEL
LIN {X 0,Y 374.636,Z 605.697,A -85,B 0,C 180,E1 -12471.99,E2 -12471.99} C_VEL
LIN {X 0,Y 374.477,Z 607.305,A -85,B 0,C 180,E1 -12473.089,E2 -12473.089} C_VEL
LIN {X 0,Y 374.349,Z 608.518,A -85,B 0,C 180,E1 -12474.409,E2 -12474.409} C_VEL
LIN {X 0,Y 374.305,Z 608.965,A -85,B 0,C 180,E1 -12475.716,E2 -12475.716} C_VEL
LIN {X 0,Y 374.34,Z 608.238,A -85,B 0,C 180,E1 -12477.656,E2 -12477.656} C_VEL
LIN {X 0,Y 374.549,Z 605.954,A -85,B 0,C 180,E1 -12479.56,E2 -12479.56} C_VEL
LIN {X 0,Y 374.764,Z 602.295,A -85,B 0,C 180,E1 -12481.343,E2 -12481.343} C_VEL
LIN {X 0,Y 375.1,Z 597.367,A -85,B 0,C 180,E1 -12482.976,E2 -12482.976} C_VEL
LIN {X 0,Y 375.467,Z 592.439,A -85,B 0,C 180,E1 -12484.246,E2 -12484.246} C_VEL
LIN {X 0,Y 375.888,Z 586.842,A -85,B 0,C 180,E1 -12485.417,E2 -12485.417} C_VEL
LIN {X 0,Y 376.456,Z 579.301,A -85,B 0,C 180,E1 -12486.701,E2 -12486.701} C_VEL
LIN {X 0,Y 377.092,Z 570.873,A -85,B 0,C 180,E1 -12487.826,E2 -12487.826} C_VEL
LIN {X 0,Y 377.555,Z 563.101,A -85,B 0,C 180,E1 -12488.667,E2 -12488.667} C_VEL
LIN {X 0,Y 378.197,Z 553.796,A -85,B 0,C 180,E1 -12489.466,E2 -12489.466} C_VEL
LIN {X 0,Y 378.017,Z 548.208,A -85,B 0,C 180,E1 -12489.882,E2 -12489.882} C_VEL
LIN {X 0,Y 376.481,Z 538.112,A -85,B 0,C 180,E1 -12490.507,E2 -12490.507} C_VEL
LIN {X 0,Y 374.849,Z 528.463,A -85,B 0,C 180,E1 -12490.988,E2 -12490.988} C_VEL
LIN {X 0,Y 375.021,Z 521.329,A -85,B 0,C 180,E1 -12494.789,E2 -12494.789} C_VEL
LIN {X 0,Y 375.254,Z 515.115,A -85,B 0,C 180,E1 -12498.111,E2 -12498.111} C_VEL
LIN {X 0,Y 375.404,Z 508.966,A -85,B 0,C 180,E1 -12501.386,E2 -12501.386} C_VEL
LIN {X 0,Y 375.6,Z 502.864,A -85,B 0,C 180,E1 -12504.631,E2 -12504.631} C_VEL
LIN {X 0,Y 375.704,Z 498.502,A -85,B 0,C 180,E1 -12506.984,E2 -12506.984} C_VEL
LIN {X 0,Y 376.434,Z 498.408,A -85,B 0,C 180,E1 -12509.999,E2 -12509.999} C_VEL
LIN {X 0,Y 376.355,Z 498.419,A -85,B 0,C 180,E1 -12512.14,E2 -12512.14} C_VEL
LIN {X 0,Y 376.249,Z 498.433,A -85,B 0,C 180,E1 -12516.434,E2 -12516.434} C_VEL
LIN {X 0,Y 376.206,Z 498.437,A -85,B 0,C 180,E1 -12518.594,E2 -12518.594} C_VEL
LIN {X 0,Y 376.05,Z 498.456,A -85,B 0,C 180,E1 -12521.863,E2 -12521.863} C_VEL
LIN {X 0,Y 376.059,Z 498.452,A -85,B 0,C 180,E1 -12525.167,E2 -12525.167} C_VEL
LIN {X 0,Y 376.024,Z 498.46,A -85,B 0,C 180,E1 -12528.525,E2 -12528.525} C_VEL
LIN {X 0,Y 375.963,Z 498.467,A -85,B 0,C 180,E1 -12531.954,E2 -12531.954} C_VEL
LIN {X 0,Y 375.99,Z 498.464,A -85,B 0,C 180,E1 -12534.15,E2 -12534.15} C_VEL
LIN {X 0,Y 375.354,Z 498.548,A -85,B 0,C 180,E1 -12535.044,E2 -12535.044} C_VEL
LIN {X 0,Y 372.549,Z 498.899,A -85,B 0,C 180,E1 -12536.5,E2 -12536.5} C_VEL
LIN {X 0,Y 370.137,Z 499.195,A -85,B 0,C 180,E1 -12537.676,E2 -12537.676} C_VEL
LIN {X 0,Y 369.065,Z 499.326,A -85,B 0,C 180,E1 -12538.586,E2 -12538.586} C_VEL
LIN {X 0,Y 368.959,Z 499.337,A -85,B 0,C 180,E1 -12538.894,E2 -12538.894} C_VEL
LIN {X 0,Y 368.899,Z 499.349,A -85,B 0,C 180,E1 -12542.237,E2 -12542.237} C_VEL
LIN {X 0,Y 368.928,Z 499.34,A -85,B 0,C 180,E1 -12545.001,E2 -12545.001} C_VEL
LIN {X 0,Y 368.909,Z 499.344,A -85,B 0,C 180,E1 -12548.64,E2 -12548.64} C_VEL
LIN {X 0,Y 368.881,Z 499.351,A -85,B 0,C 180,E1 -12552.009,E2 -12552.009} C_VEL
LIN {X 0,Y 368.955,Z 499.337,A -85,B 0,C 180,E1 -12555.187,E2 -12555.187} C_VEL
LIN {X 0,Y 368.939,Z 499.343,A -85,B 0,C 180,E1 -12558.185,E2 -12558.185} C_VEL
LIN {X 0,Y 368.911,Z 499.343,A -85,B 0,C 180,E1 -12561.358,E2 -12561.358} C_VEL
LIN {X 0,Y 368.934,Z 499.34,A -85,B 0,C 180,E1 -12565.146,E2 -12565.146} C_VEL
LIN {X 0,Y 368.926,Z 499.34,A -85,B 0,C 180,E1 -12569.046,E2 -12569.046} C_VEL
LIN {X 0,Y 368.973,Z 499.337,A -85,B 0,C 180,E1 -12571.563,E2 -12571.563} C_VEL
LIN {X 0,Y 368.997,Z 499.336,A -85,B 0,C 180,E1 -12574.02,E2 -12574.02} C_VEL
LIN {X 0,Y 368.93,Z 499.343,A -85,B 0,C 180,E1 -12577.605,E2 -12577.605} C_VEL
LIN {X 0,Y 368.98,Z 499.334,A -85,B 0,C 180,E1 -12581.107,E2 -12581.107} C_VEL
LIN {X 0,Y 368.996,Z 499.333,A -85,B 0,C 180,E1 -12584.535,E2 -12584.535} C_VEL
LIN {X 0,Y 369.011,Z 499.334,A -85,B 0,C 180,E1 -12587.907,E2 -12587.907} C_VEL
LIN {X 0,Y 369.226,Z 499.308,A -85,B 0,C 180,E1 -12591.8,E2 -12591.8} C_VEL
LIN {X 0,Y 369.142,Z 499.314,A -85,B 0,C 180,E1 -12594.537,E2 -12594.537} C_VEL
LIN {X 0,Y 369.317,Z 499.297,A -85,B 0,C 180,E1 -12597.819,E2 -12597.819} C_VEL
LIN {X 0,Y 369.456,Z 499.278,A -85,B 0,C 180,E1 -12600,E2 -12600} C_VEL
LIN {X 0,Y 369.317,Z 499.294,A -85,B 0,C 180,E1 -12602.181,E2 -12602.181} C_VEL
LIN {X 0,Y 369.206,Z 499.305,A -85,B 0,C 180,E1 -12606.558,E2 -12606.558} C_VEL
LIN {X 0,Y 369.135,Z 499.314,A -85,B 0,C 180,E1 -12608.761,E2 -12608.761} C_VEL
LIN {X 0,Y 369.003,Z 499.333,A -85,B 0,C 180,E1 -12612.093,E2 -12612.093} C_VEL
LIN {X 0,Y 368.995,Z 499.336,A -85,B 0,C 180,E1 -12615.465,E2 -12615.465} C_VEL
LIN {X 0,Y 368.955,Z 499.337,A -85,B 0,C 180,E1 -12618.894,E2 -12618.894} C_VEL
LIN {X 0,Y 368.929,Z 499.34,A -85,B 0,C 180,E1 -12622.395,E2 -12622.395} C_VEL
LIN {X 0,Y 368.997,Z 499.334,A -85,B 0,C 180,E1 -12625.98,E2 -12625.98} C_VEL
LIN {X 0,Y 368.965,Z 499.336,A -85,B 0,C 180,E1 -12628.814,E2 -12628.814} C_VEL
LIN {X 0,Y 368.907,Z 499.343,A -85,B 0,C 180,E1 -12632.237,E2 -12632.237} C_VEL
LIN {X 0,Y 368.926,Z 499.342,A -85,B 0,C 180,E1 -12635.002,E2 -12635.002} C_VEL
LIN {X 0,Y 368.907,Z 499.343,A -85,B 0,C 180,E1 -12638.641,E2 -12638.641} C_VEL
LIN {X 0,Y 368.879,Z 499.348,A -85,B 0,C 180,E1 -12642.01,E2 -12642.01} C_VEL
LIN {X 0,Y 368.924,Z 499.344,A -85,B 0,C 180,E1 -12645.183,E2 -12645.183} C_VEL
LIN {X 0,Y 368.908,Z 499.343,A -85,B 0,C 180,E1 -12648.182,E2 -12648.182} C_VEL
LIN {X 0,Y 368.912,Z 499.347,A -85,B 0,C 180,E1 -12651.359,E2 -12651.359} C_VEL
LIN {X 0,Y 368.98,Z 499.439,A -85,B 0,C 180,E1 -12653.029,E2 -12653.029} C_VEL
LIN {X 0,Y 369.969,Z 504.976,A -85,B 0,C 180,E1 -12655.918,E2 -12655.918} C_VEL
LIN {X 0,Y 370.614,Z 508.956,A -85,B 0,C 180,E1 -12657.93,E2 -12657.93} C_VEL
LIN {X 0,Y 370.093,Z 515.104,A -85,B 0,C 180,E1 -12660.872,E2 -12660.872} C_VEL
LIN {X 0,Y 369.289,Z 523.195,A -85,B 0,C 180,E1 -12664.647,E2 -12664.647} C_VEL
LIN {X 0,Y 368.661,Z 530.887,A -85,B 0,C 180,E1 -12668.178,E2 -12668.178} C_VEL
LIN {X 0,Y 368.178,Z 538.552,A -85,B 0,C 180,E1 -12671.642,E2 -12671.642} C_VEL
LIN {X 0,Y 367.87,Z 545.979,A -85,B 0,C 180,E1 -12674.984,E2 -12674.984} C_VEL
LIN {X 0,Y 369.168,Z 557.924,A -85,B 0,C 180,E1 -12675.478,E2 -12675.478} C_VEL
LIN {X 0,Y 370.108,Z 568.935,A -85,B 0,C 180,E1 -12676.121,E2 -12676.121} C_VEL
LIN {X 0,Y 370.454,Z 577.051,A -85,B 0,C 180,E1 -12676.745,E2 -12676.745} C_VEL
LIN {X 0,Y 369.835,Z 586.593,A -85,B 0,C 180,E1 -12677.656,E2 -12677.656} C_VEL
LIN {X 0,Y 369.302,Z 594.574,A -85,B 0,C 180,E1 -12678.613,E2 -12678.613} C_VEL
LIN {X 0,Y 368.796,Z 601.146,A -85,B 0,C 180,E1 -12679.57,E2 -12679.57} C_VEL
LIN {X 0,Y 368.363,Z 607.37,A -85,B 0,C 180,E1 -12680.668,E2 -12680.668} C_VEL
LIN {X 0,Y 368.016,Z 612.523,A -85,B 0,C 180,E1 -12681.766,E2 -12681.766} C_VEL
LIN {X 0,Y 367.786,Z 616.797,A -85,B 0,C 180,E1 -12682.866,E2 -12682.866} C_VEL
LIN {X 0,Y 367.568,Z 620.016,A -85,B 0,C 180,E1 -12683.854,E2 -12683.854} C_VEL
LIN {X 0,Y 367.551,Z 624.343,A -85,B 0,C 180,E1 -12685.614,E2 -12685.614} C_VEL
LIN {X 0,Y 367.438,Z 626.269,A -85,B 0,C 180,E1 -12686.711,E2 -12686.711} C_VEL
LIN {X 0,Y 367.426,Z 627.669,A -85,B 0,C 180,E1 -12687.808,E2 -12687.808} C_VEL
LIN {X 0,Y 367.469,Z 628.565,A -85,B 0,C 180,E1 -12688.905,E2 -12688.905} C_VEL
LIN {X 0,Y 367.527,Z 628.88,A -85,B 0,C 180,E1 -12690.001,E2 -12690.001} C_VEL
LIN {X 0,Y 367.468,Z 628.646,A -85,B 0,C 180,E1 -12691.096,E2 -12691.096} C_VEL
LIN {X 0,Y 367.419,Z 627.928,A -85,B 0,C 180,E1 -12692.193,E2 -12692.193} C_VEL
LIN {X 0,Y 367.429,Z 626.718,A -85,B 0,C 180,E1 -12693.29,E2 -12693.29} C_VEL
LIN {X 0,Y 367.551,Z 624.994,A -85,B 0,C 180,E1 -12694.387,E2 -12694.387} C_VEL
LIN {X 0,Y 367.549,Z 621.919,A -85,B 0,C 180,E1 -12695.775,E2 -12695.775} C_VEL
LIN {X 0,Y 367.923,Z 616.35,A -85,B 0,C 180,E1 -12697.685,E2 -12697.685} C_VEL
LIN {X 0,Y 368.465,Z 610.027,A -85,B 0,C 180,E1 -12699.331,E2 -12699.331} C_VEL
LIN {X 0,Y 369.127,Z 603.458,A -85,B 0,C 180,E1 -12700.699,E2 -12700.699} C_VEL
LIN {X 0,Y 370.037,Z 595.382,A -85,B 0,C 180,E1 -12702.06,E2 -12702.06} C_VEL
LIN {X 0,Y 370.932,Z 586.197,A -85,B 0,C 180,E1 -12703.282,E2 -12703.282} C_VEL
LIN {X 0,Y 371.697,Z 577.424,A -85,B 0,C 180,E1 -12704.23,E2 -12704.23} C_VEL
LIN {X 0,Y 371.591,Z 567.242,A -85,B 0,C 180,E1 -12705.181,E2 -12705.181} C_VEL
LIN {X 0,Y 370.498,Z 556.676,A -85,B 0,C 180,E1 -12706.036,E2 -12706.036} C_VEL
LIN {X 0,Y 368.035,Z 544.197,A -85,B 0,C 180,E1 -12706.898,E2 -12706.898} C_VEL
LIN {X 0,Y 368.579,Z 536.198,A -85,B 0,C 180,E1 -12710.881,E2 -12710.881} C_VEL
LIN {X 0,Y 369.253,Z 528.905,A -85,B 0,C 180,E1 -12714.755,E2 -12714.755} C_VEL
LIN {X 0,Y 370.044,Z 522.714,A -85,B 0,C 180,E1 -12718.347,E2 -12718.347} C_VEL
LIN {X 0,Y 370.813,Z 517.85,A -85,B 0,C 180,E1 -12721.474,E2 -12721.474} C_VEL
LIN {X 0,Y 371.214,Z 514.914,A -85,B 0,C 180,E1 -12723.589,E2 -12723.589} C_VEL
LIN {X 0,Y 371.112,Z 512.118,A -85,B 0,C 180,E1 -12725.95,E2 -12725.95} C_VEL
LIN {X 0,Y 370.666,Z 509.216,A -85,B 0,C 180,E1 -12728.979,E2 -12728.979} C_VEL
LIN {X 0,Y 370.282,Z 506.876,A -85,B 0,C 180,E1 -12732.25,E2 -12732.25} C_VEL
LIN {X 0,Y 370.003,Z 505.423,A -85,B 0,C 180,E1 -12735.349,E2 -12735.349} C_VEL
LIN {X 0,Y 369.855,Z 504.712,A -85,B 0,C 180,E1 -12738.312,E2 -12738.312} C_VEL
LIN {X 0,Y 369.825,Z 504.593,A -85,B 0,C 180,E1 -12741.183,E2 -12741.183} C_VEL
LIN {X 0,Y 369.819,Z 504.959,A -85,B 0,C 180,E1 -12743.905,E2 -12743.905} C_VEL
LIN {X 0,Y 369.872,Z 505.782,A -85,B 0,C 180,E1 -12746.726,E2 -12746.726} C_VEL
LIN {X 0,Y 369.641,Z 506.833,A -85,B 0,C 180,E1 -12749.113,E2 -12749.113} C_VEL
LIN {X 0,Y 369.34,Z 508.188,A -85,B 0,C 180,E1 -12751.594,E2 -12751.594} C_VEL
LIN {X 0,Y 368.925,Z 510.56,A -85,B 0,C 180,E1 -12755.222,E2 -12755.222} C_VEL
LIN {X 0,Y 368.617,Z 513.488,A -85,B 0,C 180,E1 -12759.105,E2 -12759.105} C_VEL
LIN {X 0,Y 368.336,Z 516.746,A -85,B 0,C 180,E1 -12762.946,E2 -12762.946} C_VEL
LIN {X 0,Y 368.318,Z 517.027,A -85,B 0,C 180,E1 -12763.263,E2 -12763.263} C_VEL
LIN {X 0,Y 372.194,Z 529.829,A -85,B 0,C 180,E1 -12764.37,E2 -12764.37} C_VEL
LIN {X 0,Y 373.704,Z 537.674,A -85,B 0,C 180,E1 -12765.113,E2 -12765.113} C_VEL
LIN {X 0,Y 372.91,Z 546.777,A -85,B 0,C 180,E1 -12765.957,E2 -12765.957} C_VEL
LIN {X 0,Y 371.916,Z 557.147,A -85,B 0,C 180,E1 -12767.171,E2 -12767.171} C_VEL
LIN {X 0,Y 371.078,Z 564.51,A -85,B 0,C 180,E1 -12768.253,E2 -12768.253} C_VEL
LIN {X 0,Y 370.402,Z 570.636,A -85,B 0,C 180,E1 -12769.339,E2 -12769.339} C_VEL
LIN {X 0,Y 369.614,Z 576.911,A -85,B 0,C 180,E1 -12770.699,E2 -12770.699} C_VEL
LIN {X 0,Y 369.14,Z 581.384,A -85,B 0,C 180,E1 -12771.902,E2 -12771.902} C_VEL
LIN {X 0,Y 368.41,Z 585.911,A -85,B 0,C 180,E1 -12773.428,E2 -12773.428} C_VEL
LIN {X 0,Y 368.237,Z 588.335,A -85,B 0,C 180,E1 -12774.524,E2 -12774.524} C_VEL
LIN {X 0,Y 368.153,Z 590.227,A -85,B 0,C 180,E1 -12775.621,E2 -12775.621} C_VEL
LIN {X 0,Y 367.903,Z 591.623,A -85,B 0,C 180,E1 -12776.715,E2 -12776.715} C_VEL
LIN {X 0,Y 367.719,Z 592.492,A -85,B 0,C 180,E1 -12777.809,E2 -12777.809} C_VEL
LIN {X 0,Y 367.59,Z 592.761,A -85,B 0,C 180,E1 -12778.905,E2 -12778.905} C_VEL
LIN {X 0,Y 367.549,Z 592.524,A -85,B 0,C 180,E1 -12780,E2 -12780} C_VEL
LIN {X 0,Y 367.559,Z 591.801,A -85,B 0,C 180,E1 -12781.096,E2 -12781.096} C_VEL
LIN {X 0,Y 367.598,Z 590.584,A -85,B 0,C 180,E1 -12782.191,E2 -12782.191} C_VEL
LIN {X 0,Y 367.654,Z 587.64,A -85,B 0,C 180,E1 -12783.836,E2 -12783.836} C_VEL
LIN {X 0,Y 367.85,Z 583.414,A -85,B 0,C 180,E1 -12785.482,E2 -12785.482} C_VEL
LIN {X 0,Y 368.222,Z 577.745,A -85,B 0,C 180,E1 -12787.126,E2 -12787.126} C_VEL
LIN {X 0,Y 368.476,Z 571.542,A -85,B 0,C 180,E1 -12788.501,E2 -12788.501} C_VEL
LIN {X 0,Y 368.861,Z 565.509,A -85,B 0,C 180,E1 -12789.597,E2 -12789.597} C_VEL
LIN {X 0,Y 369.381,Z 557.207,A -85,B 0,C 180,E1 -12790.83,E2 -12790.83} C_VEL
LIN {X 0,Y 369.946,Z 548.13,A -85,B 0,C 180,E1 -12791.923,E2 -12791.923} C_VEL
LIN {X 0,Y 370.507,Z 538.048,A -85,B 0,C 180,E1 -12792.878,E2 -12792.878} C_VEL
LIN {X 0,Y 370.732,Z 532.885,A -85,B 0,C 180,E1 -12793.28,E2 -12793.28} C_VEL
LIN {X 0,Y 368.989,Z 521.553,A -85,B 0,C 180,E1 -12794.048,E2 -12794.048} C_VEL
LIN {X 0,Y 367.696,Z 513.28,A -85,B 0,C 180,E1 -12794.494,E2 -12794.494} C_VEL
LIN {X 0,Y 367.771,Z 509.107,A -85,B 0,C 180,E1 -12797.804,E2 -12797.804} C_VEL
LIN {X 0,Y 367.852,Z 504.815,A -85,B 0,C 180,E1 -12801.285,E2 -12801.285} C_VEL
LIN {X 0,Y 368.036,Z 500.525,A -85,B 0,C 180,E1 -12804.842,E2 -12804.842} C_VEL
LIN {X 0,Y 368.139,Z 499.477,A -85,B 0,C 180,E1 -12805.817,E2 -12805.817} C_VEL
LIN {X 0,Y 368.825,Z 502.221,A -85,B 0,C 180,E1 -12807.215,E2 -12807.215} C_VEL
LIN {X 0,Y 368.703,Z 508.457,A -85,B 0,C 180,E1 -12810.307,E2 -12810.307} C_VEL
LIN {X 0,Y 368.495,Z 515.059,A -85,B 0,C 180,E1 -12813.58,E2 -12813.58} C_VEL
LIN {X 0,Y 368.311,Z 521.382,A -85,B 0,C 180,E1 -12816.732,E2 -12816.732} C_VEL
LIN {X 0,Y 368.078,Z 528.87,A -85,B 0,C 180,E1 -12820.404,E2 -12820.404} C_VEL
LIN {X 0,Y 370.185,Z 538.821,A -85,B 0,C 180,E1 -12820.919,E2 -12820.919} C_VEL
LIN {X 0,Y 371.657,Z 549.11,A -85,B 0,C 180,E1 -12821.596,E2 -12821.596} C_VEL
LIN {X 0,Y 371.928,Z 553.73,A -85,B 0,C 180,E1 -12821.961,E2 -12821.961} C_VEL
LIN {X 0,Y 371.337,Z 561.326,A -85,B 0,C 180,E1 -12822.605,E2 -12822.605} C_VEL
LIN {X 0,Y 370.811,Z 568.73,A -85,B 0,C 180,E1 -12823.378,E2 -12823.378} C_VEL
LIN {X 0,Y 370.164,Z 576.083,A -85,B 0,C 180,E1 -12824.306,E2 -12824.306} C_VEL
LIN {X 0,Y 369.412,Z 584.216,A -85,B 0,C 180,E1 -12825.569,E2 -12825.569} C_VEL
LIN {X 0,Y 368.759,Z 591.648,A -85,B 0,C 180,E1 -12827.051,E2 -12827.051} C_VEL
LIN {X 0,Y 368.278,Z 597.134,A -85,B 0,C 180,E1 -12828.459,E2 -12828.459} C_VEL
LIN {X 0,Y 367.905,Z 601.337,A -85,B 0,C 180,E1 -12829.828,E2 -12829.828} C_VEL
LIN {X 0,Y 367.703,Z 603.933,A -85,B 0,C 180,E1 -12830.895,E2 -12830.895} C_VEL
LIN {X 0,Y 367.487,Z 606.441,A -85,B 0,C 180,E1 -12832.266,E2 -12832.266} C_VEL
LIN {X 0,Y 367.327,Z 608.093,A -85,B 0,C 180,E1 -12833.621,E2 -12833.621} C_VEL
LIN {X 0,Y 367.211,Z 609.076,A -85,B 0,C 180,E1 -12835.383,E2 -12835.383} C_VEL
LIN {X 0,Y 367.224,Z 608.688,A -85,B 0,C 180,E1 -12837.361,E2 -12837.361} C_VEL
LIN {X 0,Y 367.42,Z 606.434,A -85,B 0,C 180,E1 -12839.402,E2 -12839.402} C_VEL
LIN {X 0,Y 367.617,Z 603.818,A -85,B 0,C 180,E1 -12840.823,E2 -12840.823} C_VEL
LIN {X 0,Y 367.84,Z 600.532,A -85,B 0,C 180,E1 -12842.131,E2 -12842.131} C_VEL
LIN {X 0,Y 368.246,Z 595.155,A -85,B 0,C 180,E1 -12843.766,E2 -12843.766} C_VEL
LIN {X 0,Y 368.708,Z 588.852,A -85,B 0,C 180,E1 -12845.206,E2 -12845.206} C_VEL
LIN {X 0,Y 369.251,Z 582.125,A -85,B 0,C 180,E1 -12846.44,E2 -12846.44} C_VEL
LIN {X 0,Y 369.787,Z 574.977,A -85,B 0,C 180,E1 -12847.512,E2 -12847.512} C_VEL
LIN {X 0,Y 370.449,Z 566.42,A -85,B 0,C 180,E1 -12848.554,E2 -12848.554} C_VEL
LIN {X 0,Y 371.102,Z 556.576,A -85,B 0,C 180,E1 -12849.49,E2 -12849.49} C_VEL
LIN {X 0,Y 371.285,Z 550.888,A -85,B 0,C 180,E1 -12849.935,E2 -12849.935} C_VEL
LIN {X 0,Y 369.596,Z 539.222,A -85,B 0,C 180,E1 -12850.707,E2 -12850.707} C_VEL
LIN {X 0,Y 367.812,Z 528.653,A -85,B 0,C 180,E1 -12851.225,E2 -12851.225} C_VEL
LIN {X 0,Y 367.972,Z 521.524,A -85,B 0,C 180,E1 -12855.058,E2 -12855.058} C_VEL
LIN {X 0,Y 368.194,Z 515.237,A -85,B 0,C 180,E1 -12858.438,E2 -12858.438} C_VEL
LIN {X 0,Y 368.376,Z 509.141,A -85,B 0,C 180,E1 -12861.773,E2 -12861.773} C_VEL
LIN {X 0,Y 368.601,Z 501.858,A -85,B 0,C 180,E1 -12865.625,E2 -12865.625} C_VEL
LIN {X 0,Y 368.663,Z 499.379,A -85,B 0,C 180,E1 -12866.994,E2 -12866.994} C_VEL
LIN {X 0,Y 369.383,Z 499.286,A -85,B 0,C 180,E1 -12869.999,E2 -12869.999} C_VEL
LIN {X 0,Y 369.32,Z 499.296,A -85,B 0,C 180,E1 -12872.181,E2 -12872.181} C_VEL
LIN {X 0,Y 369.21,Z 499.308,A -85,B 0,C 180,E1 -12876.558,E2 -12876.558} C_VEL
LIN {X 0,Y 369.138,Z 499.316,A -85,B 0,C 180,E1 -12878.76,E2 -12878.76} C_VEL
LIN {X 0,Y 369.006,Z 499.334,A -85,B 0,C 180,E1 -12882.093,E2 -12882.093} C_VEL
LIN {X 0,Y 368.999,Z 499.331,A -85,B 0,C 180,E1 -12885.464,E2 -12885.464} C_VEL
LIN {X 0,Y 368.983,Z 499.334,A -85,B 0,C 180,E1 -12888.892,E2 -12888.892} C_VEL
LIN {X 0,Y 368.933,Z 499.344,A -85,B 0,C 180,E1 -12892.394,E2 -12892.394} C_VEL
LIN {X 0,Y 369,Z 499.335,A -85,B 0,C 180,E1 -12895.98,E2 -12895.98} C_VEL
LIN {X 0,Y 368.959,Z 499.337,A -85,B 0,C 180,E1 -12898.894,E2 -12898.894} C_VEL
LIN {X 0,Y 368.24,Z 499.43,A -85,B 0,C 180,E1 -12899.804,E2 -12899.804} C_VEL
LIN {X 0,Y 365.367,Z 499.784,A -85,B 0,C 180,E1 -12901.284,E2 -12901.284} C_VEL
LIN {X 0,Y 362.962,Z 500.086,A -85,B 0,C 180,E1 -12902.48,E2 -12902.48} C_VEL
LIN {X 0,Y 361.932,Z 500.212,A -85,B 0,C 180,E1 -12903.406,E2 -12903.406} C_VEL
LIN {X 0,Y 361.847,Z 500.223,A -85,B 0,C 180,E1 -12903.72,E2 -12903.72} C_VEL
LIN {X 0,Y 361.864,Z 500.22,A -85,B 0,C 180,E1 -12907.223,E2 -12907.223} C_VEL
LIN {X 0,Y 361.835,Z 500.224,A -85,B 0,C 180,E1 -12910.755,E2 -12910.755} C_VEL
LIN {X 0,Y 361.862,Z 500.223,A -85,B 0,C 180,E1 -12914.361,E2 -12914.361} C_VEL
LIN {X 0,Y 361.882,Z 500.219,A -85,B 0,C 180,E1 -12917.559,E2 -12917.559} C_VEL
LIN {X 0,Y 361.873,Z 500.219,A -85,B 0,C 180,E1 -12920.972,E2 -12920.972} C_VEL
LIN {X 0,Y 361.872,Z 500.22,A -85,B 0,C 180,E1 -12924.655,E2 -12924.655} C_VEL
LIN {X 0,Y 361.835,Z 500.226,A -85,B 0,C 180,E1 -12928.37,E2 -12928.37} C_VEL
LIN {X 0,Y 361.898,Z 500.216,A -85,B 0,C 180,E1 -12930.955,E2 -12930.955} C_VEL
LIN {X 0,Y 361.951,Z 500.211,A -85,B 0,C 180,E1 -12933.475,E2 -12933.475} C_VEL
LIN {X 0,Y 361.888,Z 500.217,A -85,B 0,C 180,E1 -12937.144,E2 -12937.144} C_VEL
LIN {X 0,Y 361.918,Z 500.213,A -85,B 0,C 180,E1 -12940.724,E2 -12940.724} C_VEL
LIN {X 0,Y 361.944,Z 500.213,A -85,B 0,C 180,E1 -12944.226,E2 -12944.226} C_VEL
LIN {X 0,Y 361.997,Z 500.204,A -85,B 0,C 180,E1 -12946.528,E2 -12946.528} C_VEL
LIN {X 0,Y 362.033,Z 500.203,A -85,B 0,C 180,E1 -12949.938,E2 -12949.938} C_VEL
LIN {X 0,Y 362.148,Z 500.187,A -85,B 0,C 180,E1 -12952.192,E2 -12952.192} C_VEL
LIN {X 0,Y 362.116,Z 500.189,A -85,B 0,C 180,E1 -12954.431,E2 -12954.431} C_VEL
LIN {X 0,Y 362.281,Z 500.173,A -85,B 0,C 180,E1 -12957.776,E2 -12957.776} C_VEL
LIN {X 0,Y 362.425,Z 500.154,A -85,B 0,C 180,E1 -12960,E2 -12960} C_VEL
LIN {X 0,Y 362.281,Z 500.17,A -85,B 0,C 180,E1 -12962.223,E2 -12962.223} C_VEL
LIN {X 0,Y 362.17,Z 500.181,A -85,B 0,C 180,E1 -12966.686,E2 -12966.686} C_VEL
LIN {X 0,Y 362.072,Z 500.194,A -85,B 0,C 180,E1 -12968.933,E2 -12968.933} C_VEL
LIN {X 0,Y 361.957,Z 500.209,A -85,B 0,C 180,E1 -12972.332,E2 -12972.332} C_VEL
LIN {X 0,Y 361.959,Z 500.208,A -85,B 0,C 180,E1 -12974.62,E2 -12974.62} C_VEL
LIN {X 0,Y 361.953,Z 500.211,A -85,B 0,C 180,E1 -12978.1,E2 -12978.1} C_VEL
LIN {X 0,Y 361.889,Z 500.222,A -85,B 0,C 180,E1 -12981.653,E2 -12981.653} C_VEL
LIN {X 0,Y 361.925,Z 500.215,A -85,B 0,C 180,E1 -12985.29,E2 -12985.29} C_VEL
LIN {X 0,Y 361.92,Z 500.217,A -85,B 0,C 180,E1 -12987.778,E2 -12987.778} C_VEL
LIN {X 0,Y 361.857,Z 500.226,A -85,B 0,C 180,E1 -12991.627,E2 -12991.627} C_VEL
LIN {X 0,Y 361.872,Z 500.223,A -85,B 0,C 180,E1 -12995.345,E2 -12995.345} C_VEL
LIN {X 0,Y 361.868,Z 500.221,A -85,B 0,C 180,E1 -12999.027,E2 -12999.027} C_VEL
LIN {X 0,Y 361.834,Z 500.224,A -85,B 0,C 180,E1 -13002.829,E2 -13002.829} C_VEL
LIN {X 0,Y 361.855,Z 500.223,A -85,B 0,C 180,E1 -13005.941,E2 -13005.941} C_VEL
LIN {X 0,Y 361.87,Z 500.223,A -85,B 0,C 180,E1 -13009.238,E2 -13009.238} C_VEL
LIN {X 0,Y 361.951,Z 500.235,A -85,B 0,C 180,E1 -13012.859,E2 -13012.859} C_VEL
LIN {X 0,Y 363.079,Z 506.802,A -85,B 0,C 180,E1 -13016.339,E2 -13016.339} C_VEL
LIN {X 0,Y 363.535,Z 510.602,A -85,B 0,C 180,E1 -13018.279,E2 -13018.279} C_VEL
LIN {X 0,Y 362.976,Z 516.29,A -85,B 0,C 180,E1 -13021.05,E2 -13021.05} C_VEL
LIN {X 0,Y 362.214,Z 524.01,A -85,B 0,C 180,E1 -13024.732,E2 -13024.732} C_VEL
LIN {X 0,Y 361.56,Z 531.685,A -85,B 0,C 180,E1 -13028.327,E2 -13028.327} C_VEL
LIN {X 0,Y 361.069,Z 539.305,A -85,B 0,C 180,E1 -13031.855,E2 -13031.855} C_VEL
LIN {X 0,Y 360.788,Z 545.546,A -85,B 0,C 180,E1 -13034.718,E2 -13034.718} C_VEL
LIN {X 0,Y 361.995,Z 555.796,A -85,B 0,C 180,E1 -13035.13,E2 -13035.13} C_VEL
LIN {X 0,Y 362.821,Z 565.361,A -85,B 0,C 180,E1 -13035.662,E2 -13035.662} C_VEL
LIN {X 0,Y 363.475,Z 575.453,A -85,B 0,C 180,E1 -13036.404,E2 -13036.404} C_VEL
LIN {X 0,Y 362.891,Z 586.13,A -85,B 0,C 180,E1 -13037.416,E2 -13037.416} C_VEL
LIN {X 0,Y 362.309,Z 594.154,A -85,B 0,C 180,E1 -13038.39,E2 -13038.39} C_VEL
LIN {X 0,Y 361.776,Z 600.764,A -85,B 0,C 180,E1 -13039.366,E2 -13039.366} C_VEL
LIN {X 0,Y 361.349,Z 607.023,A -85,B 0,C 180,E1 -13040.485,E2 -13040.485} C_VEL
LIN {X 0,Y 360.971,Z 612.203,A -85,B 0,C 180,E1 -13041.604,E2 -13041.604} C_VEL
LIN {X 0,Y 360.721,Z 616.502,A -85,B 0,C 180,E1 -13042.725,E2 -13042.725} C_VEL
LIN {X 0,Y 360.468,Z 620.198,A -85,B 0,C 180,E1 -13043.901,E2 -13043.901} C_VEL
LIN {X 0,Y 360.459,Z 624.09,A -85,B 0,C 180,E1 -13045.528,E2 -13045.528} C_VEL
LIN {X 0,Y 360.358,Z 626.035,A -85,B 0,C 180,E1 -13046.646,E2 -13046.646} C_VEL
LIN {X 0,Y 360.327,Z 627.453,A -85,B 0,C 180,E1 -13047.765,E2 -13047.765} C_VEL
LIN {X 0,Y 360.369,Z 628.36,A -85,B 0,C 180,E1 -13048.883,E2 -13048.883} C_VEL
LIN {X 0,Y 360.429,Z 628.679,A -85,B 0,C 180,E1 -13050.001,E2 -13050.001} C_VEL
LIN {X 0,Y 360.368,Z 628.462,A -85,B 0,C 180,E1 -13051.118,E2 -13051.118} C_VEL
LIN {X 0,Y 360.321,Z 627.762,A -85,B 0,C 180,E1 -13052.236,E2 -13052.236} C_VEL
LIN {X 0,Y 360.35,Z 626.569,A -85,B 0,C 180,E1 -13053.355,E2 -13053.355} C_VEL
LIN {X 0,Y 360.46,Z 624.859,A -85,B 0,C 180,E1 -13054.474,E2 -13054.474} C_VEL
LIN {X 0,Y 360.46,Z 622.529,A -85,B 0,C 180,E1 -13055.595,E2 -13055.595} C_VEL
LIN {X 0,Y 360.886,Z 616.39,A -85,B 0,C 180,E1 -13057.836,E2 -13057.836} C_VEL
LIN {X 0,Y 361.47,Z 610.235,A -85,B 0,C 180,E1 -13059.513,E2 -13059.513} C_VEL
LIN {X 0,Y 362.174,Z 603.769,A -85,B 0,C 180,E1 -13060.907,E2 -13060.907} C_VEL
LIN {X 0,Y 362.911,Z 597.521,A -85,B 0,C 180,E1 -13062.016,E2 -13062.016} C_VEL
LIN {X 0,Y 363.675,Z 590.118,A -85,B 0,C 180,E1 -13063.125,E2 -13063.125} C_VEL
LIN {X 0,Y 364.91,Z 579.974,A -85,B 0,C 180,E1 -13064.358,E2 -13064.358} C_VEL
LIN {X 0,Y 364.925,Z 569.301,A -85,B 0,C 180,E1 -13065.424,E2 -13065.424} C_VEL
LIN {X 0,Y 364.357,Z 561.582,A -85,B 0,C 180,E1 -13066.098,E2 -13066.098} C_VEL
LIN {X 0,Y 362.72,Z 551.495,A -85,B 0,C 180,E1 -13066.897,E2 -13066.897} C_VEL
LIN {X 0,Y 361.057,Z 543.695,A -85,B 0,C 180,E1 -13067.487,E2 -13067.487} C_VEL
LIN {X 0,Y 361.566,Z 536.667,A -85,B 0,C 180,E1 -13071.092,E2 -13071.092} C_VEL
LIN {X 0,Y 362.327,Z 529.094,A -85,B 0,C 180,E1 -13075.261,E2 -13075.261} C_VEL
LIN {X 0,Y 363.18,Z 523.008,A -85,B 0,C 180,E1 -13078.933,E2 -13078.933} C_VEL
LIN {X 0,Y 363.892,Z 518.72,A -85,B 0,C 180,E1 -13081.811,E2 -13081.811} C_VEL
LIN {X 0,Y 364.263,Z 515.807,A -85,B 0,C 180,E1 -13084.023,E2 -13084.023} C_VEL
LIN {X 0,Y 364.188,Z 513.711,A -85,B 0,C 180,E1 -13085.855,E2 -13085.855} C_VEL
LIN {X 0,Y 363.667,Z 510.464,A -85,B 0,C 180,E1 -13089.375,E2 -13089.375} C_VEL
LIN {X 0,Y 363.319,Z 508.224,A -85,B 0,C 180,E1 -13092.687,E2 -13092.687} C_VEL
LIN {X 0,Y 363.06,Z 506.875,A -85,B 0,C 180,E1 -13095.823,E2 -13095.823} C_VEL
LIN {X 0,Y 362.91,Z 506.209,A -85,B 0,C 180,E1 -13099.049,E2 -13099.049} C_VEL
LIN {X 0,Y 362.91,Z 506.236,A -85,B 0,C 180,E1 -13102.561,E2 -13102.561} C_VEL
LIN {X 0,Y 362.891,Z 506.93,A -85,B 0,C 180,E1 -13105.831,E2 -13105.831} C_VEL
LIN {X 0,Y 362.751,Z 507.908,A -85,B 0,C 180,E1 -13108.482,E2 -13108.482} C_VEL
LIN {X 0,Y 362.456,Z 509.161,A -85,B 0,C 180,E1 -13111.004,E2 -13111.004} C_VEL
LIN {X 0,Y 361.975,Z 511.424,A -85,B 0,C 180,E1 -13114.714,E2 -13114.714} C_VEL
LIN {X 0,Y 361.647,Z 514.02,A -85,B 0,C 180,E1 -13118.332,E2 -13118.332} C_VEL
LIN {X 0,Y 361.369,Z 517.266,A -85,B 0,C 180,E1 -13122.359,E2 -13122.359} C_VEL
LIN {X 0,Y 361.379,Z 517.793,A -85,B 0,C 180,E1 -13122.724,E2 -13122.724} C_VEL
LIN {X 0,Y 365.075,Z 529.478,A -85,B 0,C 180,E1 -13123.792,E2 -13123.792} C_VEL
LIN {X 0,Y 366.908,Z 537.944,A -85,B 0,C 180,E1 -13124.636,E2 -13124.636} C_VEL
LIN {X 0,Y 367.045,Z 541.346,A -85,B 0,C 180,E1 -13124.958,E2 -13124.958} C_VEL
LIN {X 0,Y 365.935,Z 551.198,A -85,B 0,C 180,E1 -13125.968,E2 -13125.968} C_VEL
LIN {X 0,Y 365.142,Z 558.681,A -85,B 0,C 180,E1 -13126.929,E2 -13126.929} C_VEL
LIN {X 0,Y 364.251,Z 565.805,A -85,B 0,C 180,E1 -13128.029,E2 -13128.029} C_VEL
LIN {X 0,Y 363.515,Z 571.742,A -85,B 0,C 180,E1 -13129.135,E2 -13129.135} C_VEL
LIN {X 0,Y 362.679,Z 577.892,A -85,B 0,C 180,E1 -13130.52,E2 -13130.52} C_VEL
LIN {X 0,Y 361.967,Z 583.717,A -85,B 0,C 180,E1 -13132.189,E2 -13132.189} C_VEL
LIN {X 0,Y 361.299,Z 587.924,A -85,B 0,C 180,E1 -13133.858,E2 -13133.858} C_VEL
LIN {X 0,Y 361.114,Z 590.813,A -85,B 0,C 180,E1 -13135.535,E2 -13135.535} C_VEL
LIN {X 0,Y 360.859,Z 592.117,A -85,B 0,C 180,E1 -13136.651,E2 -13136.651} C_VEL
LIN {X 0,Y 360.663,Z 592.93,A -85,B 0,C 180,E1 -13137.767,E2 -13137.767} C_VEL
LIN {X 0,Y 360.528,Z 593.165,A -85,B 0,C 180,E1 -13138.883,E2 -13138.883} C_VEL
LIN {X 0,Y 360.484,Z 592.847,A -85,B 0,C 180,E1 -13140,E2 -13140} C_VEL
LIN {X 0,Y 360.479,Z 592.046,A -85,B 0,C 180,E1 -13141.117,E2 -13141.117} C_VEL
LIN {X 0,Y 360.501,Z 590.748,A -85,B 0,C 180,E1 -13142.235,E2 -13142.235} C_VEL
LIN {X 0,Y 360.577,Z 587.711,A -85,B 0,C 180,E1 -13143.912,E2 -13143.912} C_VEL
LIN {X 0,Y 360.746,Z 584.973,A -85,B 0,C 180,E1 -13145.03,E2 -13145.03} C_VEL
LIN {X 0,Y 360.9,Z 580.753,A -85,B 0,C 180,E1 -13146.389,E2 -13146.389} C_VEL
LIN {X 0,Y 361.259,Z 575.115,A -85,B 0,C 180,E1 -13147.827,E2 -13147.827} C_VEL
LIN {X 0,Y 361.625,Z 568.284,A -85,B 0,C 180,E1 -13149.226,E2 -13149.226} C_VEL
LIN {X 0,Y 362.181,Z 559.615,A -85,B 0,C 180,E1 -13150.623,E2 -13150.623} C_VEL
LIN {X 0,Y 362.755,Z 550.957,A -85,B 0,C 180,E1 -13151.738,E2 -13151.738} C_VEL
LIN {X 0,Y 363.228,Z 543.059,A -85,B 0,C 180,E1 -13152.573,E2 -13152.573} C_VEL
LIN {X 0,Y 363.653,Z 533.311,A -85,B 0,C 180,E1 -13153.41,E2 -13153.41} C_VEL
LIN {X 0,Y 361.767,Z 521.041,A -85,B 0,C 180,E1 -13154.245,E2 -13154.245} C_VEL
LIN {X 0,Y 360.623,Z 513.603,A -85,B 0,C 180,E1 -13154.648,E2 -13154.648} C_VEL
LIN {X 0,Y 360.682,Z 509.221,A -85,B 0,C 180,E1 -13158.166,E2 -13158.166} C_VEL
LIN {X 0,Y 360.783,Z 506.047,A -85,B 0,C 180,E1 -13160.765,E2 -13160.765} C_VEL
LIN {X 0,Y 360.9,Z 502.002,A -85,B 0,C 180,E1 -13164.139,E2 -13164.139} C_VEL
LIN {X 0,Y 361.082,Z 500.394,A -85,B 0,C 180,E1 -13165.662,E2 -13165.662} C_VEL
LIN {X 0,Y 361.801,Z 503.285,A -85,B 0,C 180,E1 -13167.16,E2 -13167.16} C_VEL
LIN {X 0,Y 361.682,Z 509.634,A -85,B 0,C 180,E1 -13170.346,E2 -13170.346} C_VEL
LIN {X 0,Y 361.436,Z 516.396,A -85,B 0,C 180,E1 -13173.75,E2 -13173.75} C_VEL
LIN {X 0,Y 361.245,Z 523,A -85,B 0,C 180,E1 -13177.093,E2 -13177.093} C_VEL
LIN {X 0,Y 361.054,Z 528.832,A -85,B 0,C 180,E1 -13180.039,E2 -13180.039} C_VEL
LIN {X 0,Y 363.369,Z 539.984,A -85,B 0,C 180,E1 -13180.643,E2 -13180.643} C_VEL
LIN {X 0,Y 364.888,Z 550.718,A -85,B 0,C 180,E1 -13181.387,E2 -13181.387} C_VEL
LIN {X 0,Y 364.948,Z 555.776,A -85,B 0,C 180,E1 -13181.804,E2 -13181.804} C_VEL
LIN {X 0,Y 364.112,Z 566.565,A -85,B 0,C 180,E1 -13182.821,E2 -13182.821} C_VEL
LIN {X 0,Y 363.353,Z 575.183,A -85,B 0,C 180,E1 -13183.892,E2 -13183.892} C_VEL
LIN {X 0,Y 362.668,Z 582.326,A -85,B 0,C 180,E1 -13184.982,E2 -13184.982} C_VEL
LIN {X 0,Y 362.069,Z 588.836,A -85,B 0,C 180,E1 -13186.198,E2 -13186.198} C_VEL
LIN {X 0,Y 361.483,Z 595.03,A -85,B 0,C 180,E1 -13187.629,E2 -13187.629} C_VEL
LIN {X 0,Y 360.929,Z 600.827,A -85,B 0,C 180,E1 -13189.412,E2 -13189.412} C_VEL
LIN {X 0,Y 360.562,Z 605.056,A -85,B 0,C 180,E1 -13191.231,E2 -13191.231} C_VEL
LIN {X 0,Y 360.3,Z 607.91,A -85,B 0,C 180,E1 -13193.106,E2 -13193.106} C_VEL
LIN {X 0,Y 360.123,Z 609.19,A -85,B 0,C 180,E1 -13195.05,E2 -13195.05} C_VEL
LIN {X 0,Y 360.107,Z 609.039,A -85,B 0,C 180,E1 -13197.056,E2 -13197.056} C_VEL
LIN {X 0,Y 360.182,Z 608.15,A -85,B 0,C 180,E1 -13198.208,E2 -13198.208} C_VEL
LIN {X 0,Y 360.443,Z 605.438,A -85,B 0,C 180,E1 -13200.184,E2 -13200.184} C_VEL
LIN {X 0,Y 360.669,Z 602.095,A -85,B 0,C 180,E1 -13201.708,E2 -13201.708} C_VEL
LIN {X 0,Y 360.949,Z 598.098,A -85,B 0,C 180,E1 -13203.082,E2 -13203.082} C_VEL
LIN {X 0,Y 361.352,Z 593.272,A -85,B 0,C 180,E1 -13204.395,E2 -13204.395} C_VEL
LIN {X 0,Y 361.834,Z 587.553,A -85,B 0,C 180,E1 -13205.653,E2 -13205.653} C_VEL
LIN {X 0,Y 362.37,Z 580.75,A -85,B 0,C 180,E1 -13206.874,E2 -13206.874} C_VEL
LIN {X 0,Y 363.178,Z 570.928,A -85,B 0,C 180,E1 -13208.259,E2 -13208.259} C_VEL
LIN {X 0,Y 363.742,Z 562.331,A -85,B 0,C 180,E1 -13209.204,E2 -13209.204} C_VEL
LIN {X 0,Y 364.364,Z 553.469,A -85,B 0,C 180,E1 -13209.978,E2 -13209.978} C_VEL
LIN {X 0,Y 363.599,Z 546.298,A -85,B 0,C 180,E1 -13210.523,E2 -13210.523} C_VEL
LIN {X 0,Y 362.153,Z 536.887,A -85,B 0,C 180,E1 -13211.104,E2 -13211.104} C_VEL
LIN {X 0,Y 360.761,Z 528.768,A -85,B 0,C 180,E1 -13211.507,E2 -13211.507} C_VEL
LIN {X 0,Y 360.915,Z 521.74,A -85,B 0,C 180,E1 -13215.336,E2 -13215.336} C_VEL
LIN {X 0,Y 361.13,Z 515.397,A -85,B 0,C 180,E1 -13218.777,E2 -13218.777} C_VEL
LIN {X 0,Y 361.338,Z 509.175,A -85,B 0,C 180,E1 -13222.174,E2 -13222.174} C_VEL
LIN {X 0,Y 361.57,Z 502.907,A -85,B 0,C 180,E1 -13225.54,E2 -13225.54} C_VEL
LIN {X 0,Y 361.639,Z 500.254,A -85,B 0,C 180,E1 -13227.075,E2 -13227.075} C_VEL
LIN {X 0,Y 362.333,Z 500.164,A -85,B 0,C 180,E1 -13229.999,E2 -13229.999} C_VEL
LIN {X 0,Y 362.284,Z 500.172,A -85,B 0,C 180,E1 -13232.223,E2 -13232.223} C_VEL
LIN {X 0,Y 362.174,Z 500.184,A -85,B 0,C 180,E1 -13236.686,E2 -13236.686} C_VEL
LIN {X 0,Y 362.075,Z 500.194,A -85,B 0,C 180,E1 -13238.933,E2 -13238.933} C_VEL
LIN {X 0,Y 361.961,Z 500.213,A -85,B 0,C 180,E1 -13242.332,E2 -13242.332} C_VEL
LIN {X 0,Y 361.963,Z 500.21,A -85,B 0,C 180,E1 -13244.62,E2 -13244.62} C_VEL
LIN {X 0,Y 361.96,Z 500.212,A -85,B 0,C 180,E1 -13248.099,E2 -13248.099} C_VEL
LIN {X 0,Y 361.892,Z 500.217,A -85,B 0,C 180,E1 -13251.652,E2 -13251.652} C_VEL
LIN {X 0,Y 361.928,Z 500.212,A -85,B 0,C 180,E1 -13255.289,E2 -13255.289} C_VEL
LIN {X 0,Y 361.895,Z 500.215,A -85,B 0,C 180,E1 -13258.9,E2 -13258.9} C_VEL
LIN {X 0,Y 361.837,Z 500.225,A -85,B 0,C 180,E1 -13261.629,E2 -13261.629} C_VEL
LIN {X 0,Y 361.847,Z 500.223,A -85,B 0,C 180,E1 -13263.72,E2 -13263.72} C_VEL
LIN {X 0,Y 361.172,Z 500.31,A -85,B 0,C 180,E1 -13264.648,E2 -13264.648} C_VEL
LIN {X 0,Y 358.306,Z 500.668,A -85,B 0,C 180,E1 -13266.159,E2 -13266.159} C_VEL
LIN {X 0,Y 355.888,Z 500.966,A -85,B 0,C 180,E1 -13267.38,E2 -13267.38} C_VEL
LIN {X 0,Y 354.86,Z 501.096,A -85,B 0,C 180,E1 -13268.326,E2 -13268.326} C_VEL
LIN {X 0,Y 354.781,Z 501.1,A -85,B 0,C 180,E1 -13268.646,E2 -13268.646} C_VEL
LIN {X 0,Y 354.794,Z 501.104,A -85,B 0,C 180,E1 -13272.337,E2 -13272.337} C_VEL
LIN {X 0,Y 354.851,Z 501.098,A -85,B 0,C 180,E1 -13276.117,E2 -13276.117} C_VEL
LIN {X 0,Y 354.854,Z 501.093,A -85,B 0,C 180,E1 -13279.188,E2 -13279.188} C_VEL
LIN {X 0,Y 354.807,Z 501.101,A -85,B 0,C 180,E1 -13282.402,E2 -13282.402} C_VEL
LIN {X 0,Y 354.81,Z 501.098,A -85,B 0,C 180,E1 -13284.94,E2 -13284.94} C_VEL
LIN {X 0,Y 354.791,Z 501.103,A -85,B 0,C 180,E1 -13288.405,E2 -13288.405} C_VEL
LIN {X 0,Y 354.846,Z 501.097,A -85,B 0,C 180,E1 -13291.619,E2 -13291.619} C_VEL
LIN {X 0,Y 354.896,Z 501.091,A -85,B 0,C 180,E1 -13294.172,E2 -13294.172} C_VEL
LIN {X 0,Y 354.832,Z 501.101,A -85,B 0,C 180,E1 -13297.894,E2 -13297.894} C_VEL
LIN {X 0,Y 354.92,Z 501.09,A -85,B 0,C 180,E1 -13301.891,E2 -13301.891} C_VEL
LIN {X 0,Y 354.941,Z 501.087,A -85,B 0,C 180,E1 -13305.98,E2 -13305.98} C_VEL
LIN {X 0,Y 354.98,Z 501.082,A -85,B 0,C 180,E1 -13309.736,E2 -13309.736} C_VEL
LIN {X 0,Y 355.111,Z 501.065,A -85,B 0,C 180,E1 -13312.037,E2 -13312.037} C_VEL
LIN {X 0,Y 355.09,Z 501.065,A -85,B 0,C 180,E1 -13314.321,E2 -13314.321} C_VEL
LIN {X 0,Y 355.244,Z 501.049,A -85,B 0,C 180,E1 -13317.732,E2 -13317.732} C_VEL
LIN {X 0,Y 355.395,Z 501.029,A -85,B 0,C 180,E1 -13320,E2 -13320} C_VEL
LIN {X 0,Y 355.244,Z 501.046,A -85,B 0,C 180,E1 -13322.268,E2 -13322.268} C_VEL
LIN {X 0,Y 355.136,Z 501.058,A -85,B 0,C 180,E1 -13326.819,E2 -13326.819} C_VEL
LIN {X 0,Y 355.013,Z 501.074,A -85,B 0,C 180,E1 -13329.112,E2 -13329.112} C_VEL
LIN {X 0,Y 354.918,Z 501.085,A -85,B 0,C 180,E1 -13332.581,E2 -13332.581} C_VEL
LIN {X 0,Y 354.886,Z 501.091,A -85,B 0,C 180,E1 -13336.096,E2 -13336.096} C_VEL
LIN {X 0,Y 354.898,Z 501.087,A -85,B 0,C 180,E1 -13338.472,E2 -13338.472} C_VEL
LIN {X 0,Y 354.832,Z 501.098,A -85,B 0,C 180,E1 -13342.106,E2 -13342.106} C_VEL
LIN {X 0,Y 354.896,Z 501.092,A -85,B 0,C 180,E1 -13345.828,E2 -13345.828} C_VEL
LIN {X 0,Y 354.851,Z 501.098,A -85,B 0,C 180,E1 -13349.679,E2 -13349.679} C_VEL
LIN {X 0,Y 354.827,Z 501.101,A -85,B 0,C 180,E1 -13353.682,E2 -13353.682} C_VEL
LIN {X 0,Y 354.798,Z 501.1,A -85,B 0,C 180,E1 -13356.459,E2 -13356.459} C_VEL
LIN {X 0,Y 354.821,Z 501.102,A -85,B 0,C 180,E1 -13359.424,E2 -13359.424} C_VEL
LIN {X 0,Y 354.786,Z 501.102,A -85,B 0,C 180,E1 -13362.868,E2 -13362.868} C_VEL
LIN {X 0,Y 354.799,Z 501.101,A -85,B 0,C 180,E1 -13366.11,E2 -13366.11} C_VEL
LIN {X 0,Y 354.822,Z 501.1,A -85,B 0,C 180,E1 -13369.185,E2 -13369.185} C_VEL
LIN {X 0,Y 354.899,Z 501.162,A -85,B 0,C 180,E1 -13372.756,E2 -13372.756} C_VEL
LIN {X 0,Y 356.081,Z 507.989,A -85,B 0,C 180,E1 -13376.453,E2 -13376.453} C_VEL
LIN {X 0,Y 356.503,Z 510.871,A -85,B 0,C 180,E1 -13377.961,E2 -13377.961} C_VEL
LIN {X 0,Y 355.922,Z 517.106,A -85,B 0,C 180,E1 -13381.069,E2 -13381.069} C_VEL
LIN {X 0,Y 355.117,Z 524.795,A -85,B 0,C 180,E1 -13384.818,E2 -13384.818} C_VEL
LIN {X 0,Y 354.551,Z 531.169,A -85,B 0,C 180,E1 -13387.876,E2 -13387.876} C_VEL
LIN {X 0,Y 354.03,Z 538.774,A -85,B 0,C 180,E1 -13391.481,E2 -13391.481} C_VEL
LIN {X 0,Y 353.716,Z 545.287,A -85,B 0,C 180,E1 -13394.442,E2 -13394.442} C_VEL
LIN {X 0,Y 354.948,Z 555.69,A -85,B 0,C 180,E1 -13394.864,E2 -13394.864} C_VEL
LIN {X 0,Y 355.831,Z 565.362,A -85,B 0,C 180,E1 -13395.419,E2 -13395.419} C_VEL
LIN {X 0,Y 356.429,Z 575.076,A -85,B 0,C 180,E1 -13396.148,E2 -13396.148} C_VEL
LIN {X 0,Y 356.131,Z 583.013,A -85,B 0,C 180,E1 -13396.883,E2 -13396.883} C_VEL
LIN {X 0,Y 355.376,Z 592.716,A -85,B 0,C 180,E1 -13398.016,E2 -13398.016} C_VEL
LIN {X 0,Y 354.781,Z 600.382,A -85,B 0,C 180,E1 -13399.153,E2 -13399.153} C_VEL
LIN {X 0,Y 354.301,Z 606.671,A -85,B 0,C 180,E1 -13400.294,E2 -13400.294} C_VEL
LIN {X 0,Y 353.942,Z 611.88,A -85,B 0,C 180,E1 -13401.436,E2 -13401.436} C_VEL
LIN {X 0,Y 353.655,Z 616.203,A -85,B 0,C 180,E1 -13402.579,E2 -13402.579} C_VEL
LIN {X 0,Y 353.354,Z 621.291,A -85,B 0,C 180,E1 -13404.293,E2 -13404.293} C_VEL
LIN {X 0,Y 353.369,Z 623.834,A -85,B 0,C 180,E1 -13405.438,E2 -13405.438} C_VEL
LIN {X 0,Y 353.279,Z 625.8,A -85,B 0,C 180,E1 -13406.579,E2 -13406.579} C_VEL
LIN {X 0,Y 353.233,Z 627.235,A -85,B 0,C 180,E1 -13407.72,E2 -13407.72} C_VEL
LIN {X 0,Y 353.269,Z 628.153,A -85,B 0,C 180,E1 -13408.861,E2 -13408.861} C_VEL
LIN {X 0,Y 353.331,Z 628.479,A -85,B 0,C 180,E1 -13410.001,E2 -13410.001} C_VEL
LIN {X 0,Y 353.267,Z 628.279,A -85,B 0,C 180,E1 -13411.141,E2 -13411.141} C_VEL
LIN {X 0,Y 353.226,Z 627.596,A -85,B 0,C 180,E1 -13412.281,E2 -13412.281} C_VEL
LIN {X 0,Y 353.272,Z 626.421,A -85,B 0,C 180,E1 -13413.422,E2 -13413.422} C_VEL
LIN {X 0,Y 353.374,Z 624.723,A -85,B 0,C 180,E1 -13414.563,E2 -13414.563} C_VEL
LIN {X 0,Y 353.472,Z 621.164,A -85,B 0,C 180,E1 -13416.207,E2 -13416.207} C_VEL
LIN {X 0,Y 353.826,Z 616.414,A -85,B 0,C 180,E1 -13417.993,E2 -13417.993} C_VEL
LIN {X 0,Y 354.457,Z 610.443,A -85,B 0,C 180,E1 -13419.703,E2 -13419.703} C_VEL
LIN {X 0,Y 355.23,Z 604.141,A -85,B 0,C 180,E1 -13421.122,E2 -13421.122} C_VEL
LIN {X 0,Y 356.005,Z 598.096,A -85,B 0,C 180,E1 -13422.253,E2 -13422.253} C_VEL
LIN {X 0,Y 356.807,Z 590.902,A -85,B 0,C 180,E1 -13423.382,E2 -13423.382} C_VEL
LIN {X 0,Y 357.952,Z 582.209,A -85,B 0,C 180,E1 -13424.498,E2 -13424.498} C_VEL
LIN {X 0,Y 358.27,Z 571.961,A -85,B 0,C 180,E1 -13425.621,E2 -13425.621} C_VEL
LIN {X 0,Y 357.675,Z 561.986,A -85,B 0,C 180,E1 -13426.554,E2 -13426.554} C_VEL
LIN {X 0,Y 356.046,Z 552.032,A -85,B 0,C 180,E1 -13427.392,E2 -13427.392} C_VEL
LIN {X 0,Y 354.052,Z 543.273,A -85,B 0,C 180,E1 -13428.07,E2 -13428.07} C_VEL
LIN {X 0,Y 354.545,Z 537.174,A -85,B 0,C 180,E1 -13431.305,E2 -13431.305} C_VEL
LIN {X 0,Y 355.263,Z 530.341,A -85,B 0,C 180,E1 -13435.172,E2 -13435.172} C_VEL
LIN {X 0,Y 355.982,Z 525.274,A -85,B 0,C 180,E1 -13438.283,E2 -13438.283} C_VEL
LIN {X 0,Y 356.641,Z 521.485,A -85,B 0,C 180,E1 -13440.822,E2 -13440.822} C_VEL
LIN {X 0,Y 357.21,Z 517.978,A -85,B 0,C 180,E1 -13443.429,E2 -13443.429} C_VEL
LIN {X 0,Y 357.267,Z 516.372,A -85,B 0,C 180,E1 -13444.784,E2 -13444.784} C_VEL
LIN {X 0,Y 356.999,Z 513.507,A -85,B 0,C 180,E1 -13447.61,E2 -13447.61} C_VEL
LIN {X 0,Y 356.602,Z 511.148,A -85,B 0,C 180,E1 -13450.57,E2 -13450.57} C_VEL
LIN {X 0,Y 356.302,Z 509.344,A -85,B 0,C 180,E1 -13453.66,E2 -13453.66} C_VEL
LIN {X 0,Y 356.066,Z 508.171,A -85,B 0,C 180,E1 -13456.913,E2 -13456.913} C_VEL
LIN {X 0,Y 355.961,Z 507.694,A -85,B 0,C 180,E1 -13460.355,E2 -13460.355} C_VEL
LIN {X 0,Y 355.975,Z 507.74,A -85,B 0,C 180,E1 -13462.264,E2 -13462.264} C_VEL
LIN {X 0,Y 355.948,Z 508.443,A -85,B 0,C 180,E1 -13466.024,E2 -13466.024} C_VEL
LIN {X 0,Y 355.707,Z 509.574,A -85,B 0,C 180,E1 -13469.089,E2 -13469.089} C_VEL
LIN {X 0,Y 355.213,Z 511.572,A -85,B 0,C 180,E1 -13472.931,E2 -13472.931} C_VEL
LIN {X 0,Y 354.779,Z 513.979,A -85,B 0,C 180,E1 -13476.66,E2 -13476.66} C_VEL
LIN {X 0,Y 354.614,Z 515.738,A -85,B 0,C 180,E1 -13479.1,E2 -13479.1} C_VEL
LIN {X 0,Y 354.376,Z 518.2,A -85,B 0,C 180,E1 -13482.105,E2 -13482.105} C_VEL
LIN {X 0,Y 358.043,Z 529.215,A -85,B 0,C 180,E1 -13483.171,E2 -13483.171} C_VEL
LIN {X 0,Y 359.967,Z 537.078,A -85,B 0,C 180,E1 -13483.992,E2 -13483.992} C_VEL
LIN {X 0,Y 360.604,Z 541.616,A -85,B 0,C 180,E1 -13484.481,E2 -13484.481} C_VEL
LIN {X 0,Y 359.365,Z 551.855,A -85,B 0,C 180,E1 -13485.561,E2 -13485.561} C_VEL
LIN {X 0,Y 358.371,Z 560.237,A -85,B 0,C 180,E1 -13486.678,E2 -13486.678} C_VEL
LIN {X 0,Y 357.426,Z 567.188,A -85,B 0,C 180,E1 -13487.797,E2 -13487.797} C_VEL
LIN {X 0,Y 356.432,Z 574.323,A -85,B 0,C 180,E1 -13489.204,E2 -13489.204} C_VEL
LIN {X 0,Y 355.46,Z 580.983,A -85,B 0,C 180,E1 -13490.899,E2 -13490.899} C_VEL
LIN {X 0,Y 354.756,Z 585.642,A -85,B 0,C 180,E1 -13492.46,E2 -13492.46} C_VEL
LIN {X 0,Y 354.286,Z 588.615,A -85,B 0,C 180,E1 -13493.736,E2 -13493.736} C_VEL
LIN {X 0,Y 354.077,Z 591.414,A -85,B 0,C 180,E1 -13495.446,E2 -13495.446} C_VEL
LIN {X 0,Y 353.817,Z 592.629,A -85,B 0,C 180,E1 -13496.584,E2 -13496.584} C_VEL
LIN {X 0,Y 353.609,Z 593.356,A -85,B 0,C 180,E1 -13497.722,E2 -13497.722} C_VEL
LIN {X 0,Y 353.467,Z 593.564,A -85,B 0,C 180,E1 -13498.861,E2 -13498.861} C_VEL
LIN {X 0,Y 353.403,Z 593.172,A -85,B 0,C 180,E1 -13500,E2 -13500} C_VEL
LIN {X 0,Y 353.383,Z 592.282,A -85,B 0,C 180,E1 -13501.14,E2 -13501.14} C_VEL
LIN {X 0,Y 353.404,Z 590.898,A -85,B 0,C 180,E1 -13502.28,E2 -13502.28} C_VEL
LIN {X 0,Y 353.503,Z 587.773,A -85,B 0,C 180,E1 -13503.99,E2 -13503.99} C_VEL
LIN {X 0,Y 353.664,Z 584.941,A -85,B 0,C 180,E1 -13505.131,E2 -13505.131} C_VEL
LIN {X 0,Y 353.779,Z 581.313,A -85,B 0,C 180,E1 -13506.318,E2 -13506.318} C_VEL
LIN {X 0,Y 354.172,Z 576.07,A -85,B 0,C 180,E1 -13507.698,E2 -13507.698} C_VEL
LIN {X 0,Y 354.388,Z 570.797,A -85,B 0,C 180,E1 -13508.841,E2 -13508.841} C_VEL
LIN {X 0,Y 354.817,Z 564.494,A -85,B 0,C 180,E1 -13509.981,E2 -13509.981} C_VEL
LIN {X 0,Y 355.393,Z 555.9,A -85,B 0,C 180,E1 -13511.261,E2 -13511.261} C_VEL
LIN {X 0,Y 355.98,Z 546.268,A -85,B 0,C 180,E1 -13512.398,E2 -13512.398} C_VEL
LIN {X 0,Y 356.539,Z 537.172,A -85,B 0,C 180,E1 -13513.247,E2 -13513.247} C_VEL
LIN {X 0,Y 356.325,Z 531.795,A -85,B 0,C 180,E1 -13513.691,E2 -13513.691} C_VEL
LIN {X 0,Y 354.608,Z 521.146,A -85,B 0,C 180,E1 -13514.406,E2 -13514.406} C_VEL
LIN {X 0,Y 353.554,Z 513.912,A -85,B 0,C 180,E1 -13514.812,E2 -13514.812} C_VEL
LIN {X 0,Y 353.593,Z 509.327,A -85,B 0,C 180,E1 -13518.543,E2 -13518.543} C_VEL
LIN {X 0,Y 353.73,Z 504.961,A -85,B 0,C 180,E1 -13522.179,E2 -13522.179} C_VEL
LIN {X 0,Y 353.982,Z 501.257,A -85,B 0,C 180,E1 -13525.465,E2 -13525.465} C_VEL
LIN {X 0,Y 354.785,Z 504.349,A -85,B 0,C 180,E1 -13527.104,E2 -13527.104} C_VEL
LIN {X 0,Y 354.701,Z 509.483,A -85,B 0,C 180,E1 -13529.693,E2 -13529.693} C_VEL
LIN {X 0,Y 354.424,Z 517.137,A -85,B 0,C 180,E1 -13533.608,E2 -13533.608} C_VEL
LIN {X 0,Y 354.24,Z 522.826,A -85,B 0,C 180,E1 -13536.526,E2 -13536.526} C_VEL
LIN {X 0,Y 354.018,Z 528.975,A -85,B 0,C 180,E1 -13539.67,E2 -13539.67} C_VEL
LIN {X 0,Y 356.335,Z 539.918,A -85,B 0,C 180,E1 -13540.282,E2 -13540.282} C_VEL
LIN {X 0,Y 357.991,Z 551.196,A -85,B 0,C 180,E1 -13541.086,E2 -13541.086} C_VEL
LIN {X 0,Y 358.187,Z 555.326,A -85,B 0,C 180,E1 -13541.442,E2 -13541.442} C_VEL
LIN {X 0,Y 357.422,Z 564.913,A -85,B 0,C 180,E1 -13542.331,E2 -13542.331} C_VEL
LIN {X 0,Y 356.57,Z 574.328,A -85,B 0,C 180,E1 -13543.469,E2 -13543.469} C_VEL
LIN {X 0,Y 355.777,Z 582.181,A -85,B 0,C 180,E1 -13544.671,E2 -13544.671} C_VEL
LIN {X 0,Y 355.201,Z 588.073,A -85,B 0,C 180,E1 -13545.77,E2 -13545.77} C_VEL
LIN {X 0,Y 354.742,Z 592.314,A -85,B 0,C 180,E1 -13546.698,E2 -13546.698} C_VEL
LIN {X 0,Y 354.313,Z 597.135,A -85,B 0,C 180,E1 -13547.975,E2 -13547.975} C_VEL
LIN {X 0,Y 353.945,Z 600.545,A -85,B 0,C 180,E1 -13549.06,E2 -13549.06} C_VEL
LIN {X 0,Y 353.571,Z 604.708,A -85,B 0,C 180,E1 -13550.824,E2 -13550.824} C_VEL
LIN {X 0,Y 353.272,Z 607.755,A -85,B 0,C 180,E1 -13552.727,E2 -13552.727} C_VEL
LIN {X 0,Y 353.05,Z 609.315,A -85,B 0,C 180,E1 -13554.739,E2 -13554.739} C_VEL
LIN {X 0,Y 352.993,Z 609.319,A -85,B 0,C 180,E1 -13556.742,E2 -13556.742} C_VEL
LIN {X 0,Y 353.023,Z 608.963,A -85,B 0,C 180,E1 -13557.485,E2 -13557.485} C_VEL
LIN {X 0,Y 353.155,Z 607.708,A -85,B 0,C 180,E1 -13558.84,E2 -13558.84} C_VEL
LIN {X 0,Y 353.358,Z 605.732,A -85,B 0,C 180,E1 -13560.182,E2 -13560.182} C_VEL
LIN {X 0,Y 353.55,Z 603.026,A -85,B 0,C 180,E1 -13561.504,E2 -13561.504} C_VEL
LIN {X 0,Y 353.833,Z 599.515,A -85,B 0,C 180,E1 -13562.816,E2 -13562.816} C_VEL
LIN {X 0,Y 354.266,Z 593.826,A -85,B 0,C 180,E1 -13564.438,E2 -13564.438} C_VEL
LIN {X 0,Y 354.748,Z 588.338,A -85,B 0,C 180,E1 -13565.688,E2 -13565.688} C_VEL
LIN {X 0,Y 355.177,Z 583.091,A -85,B 0,C 180,E1 -13566.687,E2 -13566.687} C_VEL
LIN {X 0,Y 355.779,Z 576.032,A -85,B 0,C 180,E1 -13567.802,E2 -13567.802} C_VEL
LIN {X 0,Y 356.381,Z 568.709,A -85,B 0,C 180,E1 -13568.754,E2 -13568.754} C_VEL
LIN {X 0,Y 356.972,Z 559.824,A -85,B 0,C 180,E1 -13569.696,E2 -13569.696} C_VEL
LIN {X 0,Y 357.353,Z 552.48,A -85,B 0,C 180,E1 -13570.318,E2 -13570.318} C_VEL
LIN {X 0,Y 355.74,Z 540.757,A -85,B 0,C 180,E1 -13571.162,E2 -13571.162} C_VEL
LIN {X 0,Y 353.836,Z 530.018,A -85,B 0,C 180,E1 -13571.715,E2 -13571.715} C_VEL
LIN {X 0,Y 353.703,Z 528.901,A -85,B 0,C 180,E1 -13571.789,E2 -13571.789} C_VEL
LIN {X 0,Y 353.875,Z 521.921,A -85,B 0,C 180,E1 -13575.625,E2 -13575.625} C_VEL
LIN {X 0,Y 354.069,Z 516.583,A -85,B 0,C 180,E1 -13578.551,E2 -13578.551} C_VEL
LIN {X 0,Y 354.262,Z 510.239,A -85,B 0,C 180,E1 -13582.017,E2 -13582.017} C_VEL
LIN {X 0,Y 354.536,Z 503.953,A -85,B 0,C 180,E1 -13585.452,E2 -13585.452} C_VEL
LIN {X 0,Y 354.595,Z 501.131,A -85,B 0,C 180,E1 -13587.088,E2 -13587.088} C_VEL
LIN {X 0,Y 355.282,Z 501.042,A -85,B 0,C 180,E1 -13589.999,E2 -13589.999} C_VEL
LIN {X 0,Y 355.247,Z 501.049,A -85,B 0,C 180,E1 -13592.267,E2 -13592.267} C_VEL
LIN {X 0,Y 355.14,Z 501.059,A -85,B 0,C 180,E1 -13596.819,E2 -13596.819} C_VEL
LIN {X 0,Y 355.016,Z 501.073,A -85,B 0,C 180,E1 -13599.112,E2 -13599.112} C_VEL
LIN {X 0,Y 354.922,Z 501.088,A -85,B 0,C 180,E1 -13602.58,E2 -13602.58} C_VEL
LIN {X 0,Y 354.89,Z 501.093,A -85,B 0,C 180,E1 -13606.095,E2 -13606.095} C_VEL
LIN {X 0,Y 354.907,Z 501.09,A -85,B 0,C 180,E1 -13608.471,E2 -13608.471} C_VEL
LIN {X 0,Y 354.835,Z 501.1,A -85,B 0,C 180,E1 -13612.105,E2 -13612.105} C_VEL
LIN {X 0,Y 354.899,Z 501.09,A -85,B 0,C 180,E1 -13615.827,E2 -13615.827} C_VEL
LIN {X 0,Y 354.854,Z 501.095,A -85,B 0,C 180,E1 -13619.678,E2 -13619.678} C_VEL
LIN {X 0,Y 354.805,Z 501.101,A -85,B 0,C 180,E1 -13623.701,E2 -13623.701} C_VEL
LIN {X 0,Y 354.798,Z 501.103,A -85,B 0,C 180,E1 -13626.459,E2 -13626.459} C_VEL
LIN {X 0,Y 354.781,Z 501.1,A -85,B 0,C 180,E1 -13628.646,E2 -13628.646} C_VEL
LIN {X 0,Y 354.132,Z 501.185,A -85,B 0,C 180,E1 -13629.594,E2 -13629.594} C_VEL
LIN {X 0,Y 351.302,Z 501.538,A -85,B 0,C 180,E1 -13631.136,E2 -13631.136} C_VEL
LIN {X 0,Y 348.888,Z 501.84,A -85,B 0,C 180,E1 -13632.384,E2 -13632.384} C_VEL
LIN {X 0,Y 347.84,Z 501.967,A -85,B 0,C 180,E1 -13633.349,E2 -13633.349} C_VEL
LIN {X 0,Y 347.749,Z 501.976,A -85,B 0,C 180,E1 -13633.676,E2 -13633.676} C_VEL
LIN {X 0,Y 347.784,Z 501.974,A -85,B 0,C 180,E1 -13636.675,E2 -13636.675} C_VEL
LIN {X 0,Y 347.783,Z 501.978,A -85,B 0,C 180,E1 -13640.165,E2 -13640.165} C_VEL
LIN {X 0,Y 347.787,Z 501.978,A -85,B 0,C 180,E1 -13644.124,E2 -13644.124} C_VEL
LIN {X 0,Y 347.736,Z 501.984,A -85,B 0,C 180,E1 -13648.086,E2 -13648.086} C_VEL
LIN {X 0,Y 347.801,Z 501.971,A -85,B 0,C 180,E1 -13650.99,E2 -13650.99} C_VEL
LIN {X 0,Y 347.829,Z 501.971,A -85,B 0,C 180,E1 -13653.607,E2 -13653.607} C_VEL
LIN {X 0,Y 347.786,Z 501.977,A -85,B 0,C 180,E1 -13656.162,E2 -13656.162} C_VEL
LIN {X 0,Y 347.815,Z 501.975,A -85,B 0,C 180,E1 -13659.909,E2 -13659.909} C_VEL
LIN {X 0,Y 347.864,Z 501.965,A -85,B 0,C 180,E1 -13662.359,E2 -13662.359} C_VEL
LIN {X 0,Y 347.895,Z 501.964,A -85,B 0,C 180,E1 -13665.971,E2 -13665.971} C_VEL
LIN {X 0,Y 347.93,Z 501.958,A -85,B 0,C 180,E1 -13669.526,E2 -13669.526} C_VEL
LIN {X 0,Y 348.072,Z 501.943,A -85,B 0,C 180,E1 -13671.875,E2 -13671.875} C_VEL
LIN {X 0,Y 348.065,Z 501.941,A -85,B 0,C 180,E1 -13674.206,E2 -13674.206} C_VEL
LIN {X 0,Y 348.206,Z 501.926,A -85,B 0,C 180,E1 -13677.686,E2 -13677.686} C_VEL
LIN {X 0,Y 348.344,Z 501.907,A -85,B 0,C 180,E1 -13680,E2 -13680} C_VEL
LIN {X 0,Y 348.206,Z 501.922,A -85,B 0,C 180,E1 -13682.313,E2 -13682.313} C_VEL
LIN {X 0,Y 348.104,Z 501.934,A -85,B 0,C 180,E1 -13686.958,E2 -13686.958} C_VEL
LIN {X 0,Y 347.965,Z 501.953,A -85,B 0,C 180,E1 -13689.298,E2 -13689.298} C_VEL
LIN {X 0,Y 347.887,Z 501.96,A -85,B 0,C 180,E1 -13692.839,E2 -13692.839} C_VEL
LIN {X 0,Y 347.836,Z 501.967,A -85,B 0,C 180,E1 -13696.431,E2 -13696.431} C_VEL
LIN {X 0,Y 347.848,Z 501.965,A -85,B 0,C 180,E1 -13698.861,E2 -13698.861} C_VEL
LIN {X 0,Y 347.771,Z 501.975,A -85,B 0,C 180,E1 -13702.579,E2 -13702.579} C_VEL
LIN {X 0,Y 347.809,Z 501.972,A -85,B 0,C 180,E1 -13705.109,E2 -13705.109} C_VEL
LIN {X 0,Y 347.809,Z 501.975,A -85,B 0,C 180,E1 -13707.694,E2 -13707.694} C_VEL
LIN {X 0,Y 347.768,Z 501.976,A -85,B 0,C 180,E1 -13710.346,E2 -13710.346} C_VEL
LIN {X 0,Y 347.745,Z 501.98,A -85,B 0,C 180,E1 -13714.044,E2 -13714.044} C_VEL
LIN {X 0,Y 347.763,Z 501.98,A -85,B 0,C 180,E1 -13717.321,E2 -13717.321} C_VEL
LIN {X 0,Y 347.73,Z 501.981,A -85,B 0,C 180,E1 -13720.297,E2 -13720.297} C_VEL
LIN {X 0,Y 347.721,Z 501.986,A -85,B 0,C 180,E1 -13723.408,E2 -13723.408} C_VEL
LIN {X 0,Y 347.766,Z 501.976,A -85,B 0,C 180,E1 -13726.679,E2 -13726.679} C_VEL
LIN {X 0,Y 347.756,Z 501.977,A -85,B 0,C 180,E1 -13730.171,E2 -13730.171} C_VEL
LIN {X 0,Y 347.878,Z 502.129,A -85,B 0,C 180,E1 -13732.695,E2 -13732.695} C_VEL
LIN {X 0,Y 349.029,Z 508.827,A -85,B 0,C 180,E1 -13736.395,E2 -13736.395} C_VEL
LIN {X 0,Y 349.424,Z 511.157,A -85,B 0,C 180,E1 -13737.645,E2 -13737.645} C_VEL
LIN {X 0,Y 348.967,Z 516.787,A -85,B 0,C 180,E1 -13740.526,E2 -13740.526} C_VEL
LIN {X 0,Y 348.134,Z 524.284,A -85,B 0,C 180,E1 -13744.277,E2 -13744.277} C_VEL
LIN {X 0,Y 347.43,Z 531.911,A -85,B 0,C 180,E1 -13748.025,E2 -13748.025} C_VEL
LIN {X 0,Y 346.89,Z 539.598,A -85,B 0,C 180,E1 -13751.759,E2 -13751.759} C_VEL
LIN {X 0,Y 346.671,Z 544.459,A -85,B 0,C 180,E1 -13754.117,E2 -13754.117} C_VEL
LIN {X 0,Y 348.064,Z 556.727,A -85,B 0,C 180,E1 -13754.651,E2 -13754.651} C_VEL
LIN {X 0,Y 349.024,Z 568.173,A -85,B 0,C 180,E1 -13755.354,E2 -13755.354} C_VEL
LIN {X 0,Y 349.482,Z 578.036,A -85,B 0,C 180,E1 -13756.185,E2 -13756.185} C_VEL
LIN {X 0,Y 348.905,Z 586.422,A -85,B 0,C 180,E1 -13757.051,E2 -13757.051} C_VEL
LIN {X 0,Y 348.267,Z 594.33,A -85,B 0,C 180,E1 -13758.063,E2 -13758.063} C_VEL
LIN {X 0,Y 347.644,Z 601.695,A -85,B 0,C 180,E1 -13759.223,E2 -13759.223} C_VEL
LIN {X 0,Y 347.07,Z 609.142,A -85,B 0,C 180,E1 -13760.678,E2 -13760.678} C_VEL
LIN {X 0,Y 346.665,Z 614.946,A -85,B 0,C 180,E1 -13762.135,E2 -13762.135} C_VEL
LIN {X 0,Y 346.346,Z 619.496,A -85,B 0,C 180,E1 -13763.593,E2 -13763.593} C_VEL
LIN {X 0,Y 346.279,Z 623.578,A -85,B 0,C 180,E1 -13765.344,E2 -13765.344} C_VEL
LIN {X 0,Y 346.203,Z 625.564,A -85,B 0,C 180,E1 -13766.509,E2 -13766.509} C_VEL
LIN {X 0,Y 346.141,Z 627.017,A -85,B 0,C 180,E1 -13767.673,E2 -13767.673} C_VEL
LIN {X 0,Y 346.169,Z 627.945,A -85,B 0,C 180,E1 -13768.837,E2 -13768.837} C_VEL
LIN {X 0,Y 346.234,Z 628.278,A -85,B 0,C 180,E1 -13770.001,E2 -13770.001} C_VEL
LIN {X 0,Y 346.167,Z 628.095,A -85,B 0,C 180,E1 -13771.164,E2 -13771.164} C_VEL
LIN {X 0,Y 346.135,Z 627.43,A -85,B 0,C 180,E1 -13772.328,E2 -13772.328} C_VEL
LIN {X 0,Y 346.197,Z 626.275,A -85,B 0,C 180,E1 -13773.492,E2 -13773.492} C_VEL
LIN {X 0,Y 346.287,Z 624.592,A -85,B 0,C 180,E1 -13774.657,E2 -13774.657} C_VEL
LIN {X 0,Y 346.454,Z 620.502,A -85,B 0,C 180,E1 -13776.568,E2 -13776.568} C_VEL
LIN {X 0,Y 346.97,Z 614.74,A -85,B 0,C 180,E1 -13778.739,E2 -13778.739} C_VEL
LIN {X 0,Y 347.644,Z 609.565,A -85,B 0,C 180,E1 -13780.189,E2 -13780.189} C_VEL
LIN {X 0,Y 348.486,Z 603.174,A -85,B 0,C 180,E1 -13781.635,E2 -13781.635} C_VEL
LIN {X 0,Y 349.341,Z 597.017,A -85,B 0,C 180,E1 -13782.786,E2 -13782.786} C_VEL
LIN {X 0,Y 350.169,Z 589.732,A -85,B 0,C 180,E1 -13783.937,E2 -13783.937} C_VEL
LIN {X 0,Y 351.422,Z 581.013,A -85,B 0,C 180,E1 -13785.07,E2 -13785.07} C_VEL
LIN {X 0,Y 351.647,Z 570.415,A -85,B 0,C 180,E1 -13786.249,E2 -13786.249} C_VEL
LIN {X 0,Y 350.783,Z 560.709,A -85,B 0,C 180,E1 -13787.189,E2 -13787.189} C_VEL
LIN {X 0,Y 348.922,Z 550.501,A -85,B 0,C 180,E1 -13788.101,E2 -13788.101} C_VEL
LIN {X 0,Y 347.079,Z 542.759,A -85,B 0,C 180,E1 -13788.75,E2 -13788.75} C_VEL
LIN {X 0,Y 347.519,Z 537.708,A -85,B 0,C 180,E1 -13791.523,E2 -13791.523} C_VEL
LIN {X 0,Y 348.372,Z 530.565,A -85,B 0,C 180,E1 -13795.706,E2 -13795.706} C_VEL
LIN {X 0,Y 349.145,Z 525.597,A -85,B 0,C 180,E1 -13798.889,E2 -13798.889} C_VEL
LIN {X 0,Y 349.824,Z 521.899,A -85,B 0,C 180,E1 -13801.49,E2 -13801.49} C_VEL
LIN {X 0,Y 350.326,Z 518.519,A -85,B 0,C 180,E1 -13804.175,E2 -13804.175} C_VEL
LIN {X 0,Y 350.136,Z 515.575,A -85,B 0,C 180,E1 -13807.026,E2 -13807.026} C_VEL
LIN {X 0,Y 349.738,Z 512.968,A -85,B 0,C 180,E1 -13810.217,E2 -13810.217} C_VEL
LIN {X 0,Y 349.408,Z 510.974,A -85,B 0,C 180,E1 -13813.606,E2 -13813.606} C_VEL
LIN {X 0,Y 349.168,Z 509.8,A -85,B 0,C 180,E1 -13816.816,E2 -13816.816} C_VEL
LIN {X 0,Y 349.046,Z 509.292,A -85,B 0,C 180,E1 -13819.919,E2 -13819.919} C_VEL
LIN {X 0,Y 349,Z 509.336,A -85,B 0,C 180,E1 -13822.834,E2 -13822.834} C_VEL
LIN {X 0,Y 349.007,Z 509.822,A -85,B 0,C 180,E1 -13825.678,E2 -13825.678} C_VEL
LIN {X 0,Y 348.837,Z 510.695,A -85,B 0,C 180,E1 -13828.411,E2 -13828.411} C_VEL
LIN {X 0,Y 348.451,Z 511.887,A -85,B 0,C 180,E1 -13831.049,E2 -13831.049} C_VEL
LIN {X 0,Y 348.125,Z 513.29,A -85,B 0,C 180,E1 -13833.632,E2 -13833.632} C_VEL
LIN {X 0,Y 347.695,Z 515.711,A -85,B 0,C 180,E1 -13837.415,E2 -13837.415} C_VEL
LIN {X 0,Y 347.504,Z 517.489,A -85,B 0,C 180,E1 -13839.891,E2 -13839.891} C_VEL
LIN {X 0,Y 347.408,Z 518.809,A -85,B 0,C 180,E1 -13841.447,E2 -13841.447} C_VEL
LIN {X 0,Y 351.047,Z 529.255,A -85,B 0,C 180,E1 -13842.524,E2 -13842.524} C_VEL
LIN {X 0,Y 353.31,Z 537.937,A -85,B 0,C 180,E1 -13843.5,E2 -13843.5} C_VEL
LIN {X 0,Y 354.087,Z 542.77,A -85,B 0,C 180,E1 -13844.045,E2 -13844.045} C_VEL
LIN {X 0,Y 352.828,Z 552.747,A -85,B 0,C 180,E1 -13845.14,E2 -13845.14} C_VEL
LIN {X 0,Y 351.9,Z 560.044,A -85,B 0,C 180,E1 -13846.134,E2 -13846.134} C_VEL
LIN {X 0,Y 350.867,Z 567.023,A -85,B 0,C 180,E1 -13847.271,E2 -13847.271} C_VEL
LIN {X 0,Y 349.957,Z 572.869,A -85,B 0,C 180,E1 -13848.415,E2 -13848.415} C_VEL
LIN {X 0,Y 349.217,Z 577.81,A -85,B 0,C 180,E1 -13849.565,E2 -13849.565} C_VEL
LIN {X 0,Y 348.402,Z 583.054,A -85,B 0,C 180,E1 -13851.065,E2 -13851.065} C_VEL
LIN {X 0,Y 347.732,Z 586.691,A -85,B 0,C 180,E1 -13852.38,E2 -13852.38} C_VEL
LIN {X 0,Y 347.275,Z 589.349,A -85,B 0,C 180,E1 -13853.609,E2 -13853.609} C_VEL
LIN {X 0,Y 347.043,Z 592.022,A -85,B 0,C 180,E1 -13855.354,E2 -13855.354} C_VEL
LIN {X 0,Y 346.758,Z 593.14,A -85,B 0,C 180,E1 -13856.514,E2 -13856.514} C_VEL
LIN {X 0,Y 346.539,Z 593.778,A -85,B 0,C 180,E1 -13857.675,E2 -13857.675} C_VEL
LIN {X 0,Y 346.39,Z 593.928,A -85,B 0,C 180,E1 -13858.838,E2 -13858.838} C_VEL
LIN {X 0,Y 346.324,Z 593.491,A -85,B 0,C 180,E1 -13860,E2 -13860} C_VEL
LIN {X 0,Y 346.288,Z 592.507,A -85,B 0,C 180,E1 -13861.163,E2 -13861.163} C_VEL
LIN {X 0,Y 346.323,Z 590.141,A -85,B 0,C 180,E1 -13862.908,E2 -13862.908} C_VEL
LIN {X 0,Y 346.53,Z 586.451,A -85,B 0,C 180,E1 -13864.653,E2 -13864.653} C_VEL
LIN {X 0,Y 346.66,Z 581.812,A -85,B 0,C 180,E1 -13866.246,E2 -13866.246} C_VEL
LIN {X 0,Y 347.069,Z 576.987,A -85,B 0,C 180,E1 -13867.563,E2 -13867.563} C_VEL
LIN {X 0,Y 347.354,Z 570.395,A -85,B 0,C 180,E1 -13869.022,E2 -13869.022} C_VEL
LIN {X 0,Y 347.919,Z 562.249,A -85,B 0,C 180,E1 -13870.475,E2 -13870.475} C_VEL
LIN {X 0,Y 348.591,Z 552.836,A -85,B 0,C 180,E1 -13871.779,E2 -13871.779} C_VEL
LIN {X 0,Y 349.025,Z 545.176,A -85,B 0,C 180,E1 -13872.649,E2 -13872.649} C_VEL
LIN {X 0,Y 349.554,Z 535.786,A -85,B 0,C 180,E1 -13873.517,E2 -13873.517} C_VEL
LIN {X 0,Y 348.837,Z 529.904,A -85,B 0,C 180,E1 -13873.991,E2 -13873.991} C_VEL
LIN {X 0,Y 347.218,Z 519.455,A -85,B 0,C 180,E1 -13874.678,E2 -13874.678} C_VEL
LIN {X 0,Y 346.47,Z 514.24,A -85,B 0,C 180,E1 -13874.959,E2 -13874.959} C_VEL
LIN {X 0,Y 346.532,Z 510.883,A -85,B 0,C 180,E1 -13877.711,E2 -13877.711} C_VEL
LIN {X 0,Y 346.648,Z 506.488,A -85,B 0,C 180,E1 -13881.404,E2 -13881.404} C_VEL
LIN {X 0,Y 346.9,Z 502.153,A -85,B 0,C 180,E1 -13885.259,E2 -13885.259} C_VEL
LIN {X 0,Y 347.797,Z 505.834,A -85,B 0,C 180,E1 -13887.236,E2 -13887.236} C_VEL
LIN {X 0,Y 347.638,Z 511.899,A -85,B 0,C 180,E1 -13890.359,E2 -13890.359} C_VEL
LIN {X 0,Y 347.368,Z 518.866,A -85,B 0,C 180,E1 -13893.95,E2 -13893.95} C_VEL
LIN {X 0,Y 347.137,Z 525.499,A -85,B 0,C 180,E1 -13897.4,E2 -13897.4} C_VEL
LIN {X 0,Y 347.023,Z 529.114,A -85,B 0,C 180,E1 -13899.274,E2 -13899.274} C_VEL
LIN {X 0,Y 349.624,Z 541.362,A -85,B 0,C 180,E1 -13899.992,E2 -13899.992} C_VEL
LIN {X 0,Y 351.035,Z 551.182,A -85,B 0,C 180,E1 -13900.725,E2 -13900.725} C_VEL
LIN {X 0,Y 351.272,Z 556.891,A -85,B 0,C 180,E1 -13901.227,E2 -13901.227} C_VEL
LIN {X 0,Y 350.425,Z 567.122,A -85,B 0,C 180,E1 -13902.246,E2 -13902.246} C_VEL
LIN {X 0,Y 349.564,Z 575.626,A -85,B 0,C 180,E1 -13903.344,E2 -13903.344} C_VEL
LIN {X 0,Y 348.945,Z 581.723,A -85,B 0,C 180,E1 -13904.294,E2 -13904.294} C_VEL
LIN {X 0,Y 348.257,Z 587.999,A -85,B 0,C 180,E1 -13905.47,E2 -13905.47} C_VEL
LIN {X 0,Y 347.664,Z 593.387,A -85,B 0,C 180,E1 -13906.697,E2 -13906.697} C_VEL
LIN {X 0,Y 347.193,Z 598.324,A -85,B 0,C 180,E1 -13908.087,E2 -13908.087} C_VEL
LIN {X 0,Y 346.747,Z 602.467,A -85,B 0,C 180,E1 -13909.564,E2 -13909.564} C_VEL
LIN {X 0,Y 346.435,Z 605.576,A -85,B 0,C 180,E1 -13911.031,E2 -13911.031} C_VEL
LIN {X 0,Y 346.205,Z 607.759,A -85,B 0,C 180,E1 -13912.482,E2 -13912.482} C_VEL
LIN {X 0,Y 345.974,Z 609.41,A -85,B 0,C 180,E1 -13914.346,E2 -13914.346} C_VEL
LIN {X 0,Y 345.909,Z 609.599,A -85,B 0,C 180,E1 -13916.41,E2 -13916.41} C_VEL
LIN {X 0,Y 346.013,Z 608.262,A -85,B 0,C 180,E1 -13918.548,E2 -13918.548} C_VEL
LIN {X 0,Y 346.272,Z 606.018,A -85,B 0,C 180,E1 -13920.177,E2 -13920.177} C_VEL
LIN {X 0,Y 346.46,Z 603.33,A -85,B 0,C 180,E1 -13921.529,E2 -13921.529} C_VEL
LIN {X 0,Y 346.8,Z 599.161,A -85,B 0,C 180,E1 -13923.084,E2 -13923.084} C_VEL
LIN {X 0,Y 347.204,Z 594.195,A -85,B 0,C 180,E1 -13924.523,E2 -13924.523} C_VEL
LIN {X 0,Y 347.721,Z 588.563,A -85,B 0,C 180,E1 -13925.836,E2 -13925.836} C_VEL
LIN {X 0,Y 348.153,Z 583.529,A -85,B 0,C 180,E1 -13926.818,E2 -13926.818} C_VEL
LIN {X 0,Y 348.772,Z 576.479,A -85,B 0,C 180,E1 -13927.962,E2 -13927.962} C_VEL
LIN {X 0,Y 349.383,Z 569.257,A -85,B 0,C 180,E1 -13928.926,E2 -13928.926} C_VEL
LIN {X 0,Y 350.007,Z 560.431,A -85,B 0,C 180,E1 -13929.887,E2 -13929.887} C_VEL
LIN {X 0,Y 350.384,Z 553.27,A -85,B 0,C 180,E1 -13930.515,E2 -13930.515} C_VEL
LIN {X 0,Y 348.851,Z 542.126,A -85,B 0,C 180,E1 -13931.363,E2 -13931.363} C_VEL
LIN {X 0,Y 346.922,Z 530.708,A -85,B 0,C 180,E1 -13931.975,E2 -13931.975} C_VEL
LIN {X 0,Y 346.651,Z 529.04,A -85,B 0,C 180,E1 -13932.08,E2 -13932.08} C_VEL
LIN {X 0,Y 346.839,Z 522.103,A -85,B 0,C 180,E1 -13935.927,E2 -13935.927} C_VEL
LIN {X 0,Y 347.053,Z 515.628,A -85,B 0,C 180,E1 -13939.498,E2 -13939.498} C_VEL
LIN {X 0,Y 347.288,Z 509.178,A -85,B 0,C 180,E1 -13943.025,E2 -13943.025} C_VEL
LIN {X 0,Y 347.46,Z 503.983,A -85,B 0,C 180,E1 -13945.94,E2 -13945.94} C_VEL
LIN {X 0,Y 347.545,Z 502.009,A -85,B 0,C 180,E1 -13947.102,E2 -13947.102} C_VEL
LIN {X 0,Y 348.233,Z 501.92,A -85,B 0,C 180,E1 -13949.999,E2 -13949.999} C_VEL
LIN {X 0,Y 348.21,Z 501.926,A -85,B 0,C 180,E1 -13952.313,E2 -13952.313} C_VEL
LIN {X 0,Y 348.108,Z 501.934,A -85,B 0,C 180,E1 -13956.957,E2 -13956.957} C_VEL
LIN {X 0,Y 347.968,Z 501.95,A -85,B 0,C 180,E1 -13959.298,E2 -13959.298} C_VEL
LIN {X 0,Y 347.891,Z 501.961,A -85,B 0,C 180,E1 -13962.839,E2 -13962.839} C_VEL
LIN {X 0,Y 347.84,Z 501.971,A -85,B 0,C 180,E1 -13966.431,E2 -13966.431} C_VEL
LIN {X 0,Y 347.856,Z 501.965,A -85,B 0,C 180,E1 -13968.86,E2 -13968.86} C_VEL
LIN {X 0,Y 347.774,Z 501.977,A -85,B 0,C 180,E1 -13972.579,E2 -13972.579} C_VEL
LIN {X 0,Y 347.812,Z 501.97,A -85,B 0,C 180,E1 -13975.108,E2 -13975.108} C_VEL
LIN {X 0,Y 347.812,Z 501.971,A -85,B 0,C 180,E1 -13977.693,E2 -13977.693} C_VEL
LIN {X 0,Y 347.764,Z 501.98,A -85,B 0,C 180,E1 -13980.346,E2 -13980.346} C_VEL
LIN {X 0,Y 347.743,Z 501.981,A -85,B 0,C 180,E1 -13984.463,E2 -13984.463} C_VEL
LIN {X 0,Y 347.773,Z 501.98,A -85,B 0,C 180,E1 -13987.988,E2 -13987.988} C_VEL
LIN {X 0,Y 347.75,Z 501.981,A -85,B 0,C 180,E1 -13991.83,E2 -13991.83} C_VEL
LIN {X 0,Y 347.749,Z 501.976,A -85,B 0,C 180,E1 -13993.676,E2 -13993.676} C_VEL
LIN {X 0,Y 347.069,Z 502.064,A -85,B 0,C 180,E1 -13994.643,E2 -13994.643} C_VEL
LIN {X 0,Y 344.226,Z 502.421,A -85,B 0,C 180,E1 -13996.217,E2 -13996.217} C_VEL
LIN {X 0,Y 341.828,Z 502.719,A -85,B 0,C 180,E1 -13997.491,E2 -13997.491} C_VEL
LIN {X 0,Y 340.804,Z 502.845,A -85,B 0,C 180,E1 -13998.477,E2 -13998.477} C_VEL
LIN {X 0,Y 340.722,Z 502.853,A -85,B 0,C 180,E1 -13998.81,E2 -13998.81} C_VEL
LIN {X 0,Y 340.737,Z 502.855,A -85,B 0,C 180,E1 -14001.773,E2 -14001.773} C_VEL
LIN {X 0,Y 340.72,Z 502.855,A -85,B 0,C 180,E1 -14005.595,E2 -14005.595} C_VEL
LIN {X 0,Y 340.701,Z 502.855,A -85,B 0,C 180,E1 -14008.956,E2 -14008.956} C_VEL
LIN {X 0,Y 340.775,Z 502.848,A -85,B 0,C 180,E1 -14012.474,E2 -14012.474} C_VEL
LIN {X 0,Y 340.753,Z 502.852,A -85,B 0,C 180,E1 -14015.638,E2 -14015.638} C_VEL
LIN {X 0,Y 340.745,Z 502.852,A -85,B 0,C 180,E1 -14019.474,E2 -14019.474} C_VEL
LIN {X 0,Y 340.855,Z 502.842,A -85,B 0,C 180,E1 -14021.984,E2 -14021.984} C_VEL
LIN {X 0,Y 340.866,Z 502.839,A -85,B 0,C 180,E1 -14025.705,E2 -14025.705} C_VEL
LIN {X 0,Y 340.872,Z 502.835,A -85,B 0,C 180,E1 -14029.306,E2 -14029.306} C_VEL
LIN {X 0,Y 341.073,Z 502.809,A -85,B 0,C 180,E1 -14032.898,E2 -14032.898} C_VEL
LIN {X 0,Y 341.168,Z 502.802,A -85,B 0,C 180,E1 -14037.639,E2 -14037.639} C_VEL
LIN {X 0,Y 341.294,Z 502.785,A -85,B 0,C 180,E1 -14040,E2 -14040} C_VEL
LIN {X 0,Y 341.168,Z 502.798,A -85,B 0,C 180,E1 -14042.361,E2 -14042.361} C_VEL
LIN {X 0,Y 341.073,Z 502.81,A -85,B 0,C 180,E1 -14047.102,E2 -14047.102} C_VEL
LIN {X 0,Y 340.869,Z 502.835,A -85,B 0,C 180,E1 -14050.694,E2 -14050.694} C_VEL
LIN {X 0,Y 340.86,Z 502.837,A -85,B 0,C 180,E1 -14054.325,E2 -14054.325} C_VEL
LIN {X 0,Y 340.834,Z 502.839,A -85,B 0,C 180,E1 -14058.466,E2 -14058.466} C_VEL
LIN {X 0,Y 340.75,Z 502.853,A -85,B 0,C 180,E1 -14061.857,E2 -14061.857} C_VEL
LIN {X 0,Y 340.77,Z 502.852,A -85,B 0,C 180,E1 -14065.664,E2 -14065.664} C_VEL
LIN {X 0,Y 340.739,Z 502.851,A -85,B 0,C 180,E1 -14068.32,E2 -14068.32} C_VEL
LIN {X 0,Y 340.713,Z 502.855,A -85,B 0,C 180,E1 -14071.043,E2 -14071.043} C_VEL
LIN {X 0,Y 340.716,Z 502.857,A -85,B 0,C 180,E1 -14075.279,E2 -14075.279} C_VEL
LIN {X 0,Y 340.709,Z 502.855,A -85,B 0,C 180,E1 -14078.387,E2 -14078.387} C_VEL
LIN {X 0,Y 340.696,Z 502.857,A -85,B 0,C 180,E1 -14082.046,E2 -14082.046} C_VEL
LIN {X 0,Y 340.695,Z 502.862,A -85,B 0,C 180,E1 -14085.464,E2 -14085.464} C_VEL
LIN {X 0,Y 340.702,Z 502.856,A -85,B 0,C 180,E1 -14088.694,E2 -14088.694} C_VEL
LIN {X 0,Y 340.813,Z 502.91,A -85,B 0,C 180,E1 -14092.532,E2 -14092.532} C_VEL
LIN {X 0,Y 341.977,Z 509.579,A -85,B 0,C 180,E1 -14096.298,E2 -14096.298} C_VEL
LIN {X 0,Y 342.377,Z 512.218,A -85,B 0,C 180,E1 -14097.745,E2 -14097.745} C_VEL
LIN {X 0,Y 341.91,Z 517.378,A -85,B 0,C 180,E1 -14100.442,E2 -14100.442} C_VEL
LIN {X 0,Y 341.045,Z 525.027,A -85,B 0,C 180,E1 -14104.358,E2 -14104.358} C_VEL
LIN {X 0,Y 340.288,Z 532.946,A -85,B 0,C 180,E1 -14108.34,E2 -14108.34} C_VEL
LIN {X 0,Y 339.77,Z 540.445,A -85,B 0,C 180,E1 -14112.08,E2 -14112.08} C_VEL
LIN {X 0,Y 339.605,Z 543.925,A -85,B 0,C 180,E1 -14113.816,E2 -14113.816} C_VEL
LIN {X 0,Y 340.971,Z 555.627,A -85,B 0,C 180,E1 -14114.324,E2 -14114.324} C_VEL
LIN {X 0,Y 341.823,Z 565.225,A -85,B 0,C 180,E1 -14114.903,E2 -14114.903} C_VEL
LIN {X 0,Y 342.451,Z 575.828,A -85,B 0,C 180,E1 -14115.744,E2 -14115.744} C_VEL
LIN {X 0,Y 341.961,Z 585.886,A -85,B 0,C 180,E1 -14116.784,E2 -14116.784} C_VEL
LIN {X 0,Y 341.274,Z 593.851,A -85,B 0,C 180,E1 -14117.815,E2 -14117.815} C_VEL
LIN {X 0,Y 340.819,Z 599.571,A -85,B 0,C 180,E1 -14118.703,E2 -14118.703} C_VEL
LIN {X 0,Y 340.251,Z 605.93,A -85,B 0,C 180,E1 -14119.889,E2 -14119.889} C_VEL
LIN {X 0,Y 339.84,Z 611.201,A -85,B 0,C 180,E1 -14121.078,E2 -14121.078} C_VEL
LIN {X 0,Y 339.537,Z 615.581,A -85,B 0,C 180,E1 -14122.268,E2 -14122.268} C_VEL
LIN {X 0,Y 339.208,Z 620.719,A -85,B 0,C 180,E1 -14124.054,E2 -14124.054} C_VEL
LIN {X 0,Y 339.141,Z 624.452,A -85,B 0,C 180,E1 -14125.841,E2 -14125.841} C_VEL
LIN {X 0,Y 339.054,Z 626.793,A -85,B 0,C 180,E1 -14127.625,E2 -14127.625} C_VEL
LIN {X 0,Y 339.07,Z 627.73,A -85,B 0,C 180,E1 -14128.813,E2 -14128.813} C_VEL
LIN {X 0,Y 339.136,Z 628.075,A -85,B 0,C 180,E1 -14130.001,E2 -14130.001} C_VEL
LIN {X 0,Y 339.067,Z 627.914,A -85,B 0,C 180,E1 -14131.188,E2 -14131.188} C_VEL
LIN {X 0,Y 339.048,Z 627.272,A -85,B 0,C 180,E1 -14132.377,E2 -14132.377} C_VEL
LIN {X 0,Y 339.123,Z 626.138,A -85,B 0,C 180,E1 -14133.565,E2 -14133.565} C_VEL
LIN {X 0,Y 339.201,Z 624.466,A -85,B 0,C 180,E1 -14134.755,E2 -14134.755} C_VEL
LIN {X 0,Y 339.467,Z 619.514,A -85,B 0,C 180,E1 -14137.136,E2 -14137.136} C_VEL
LIN {X 0,Y 339.965,Z 614.916,A -85,B 0,C 180,E1 -14138.92,E2 -14138.92} C_VEL
LIN {X 0,Y 340.823,Z 608.692,A -85,B 0,C 180,E1 -14140.696,E2 -14140.696} C_VEL
LIN {X 0,Y 341.801,Z 602.248,A -85,B 0,C 180,E1 -14142.167,E2 -14142.167} C_VEL
LIN {X 0,Y 342.723,Z 596.071,A -85,B 0,C 180,E1 -14143.339,E2 -14143.339} C_VEL
LIN {X 0,Y 343.347,Z 590.718,A -85,B 0,C 180,E1 -14144.22,E2 -14144.22} C_VEL
LIN {X 0,Y 344.542,Z 583.387,A -85,B 0,C 180,E1 -14145.227,E2 -14145.227} C_VEL
LIN {X 0,Y 344.966,Z 574.386,A -85,B 0,C 180,E1 -14146.317,E2 -14146.317} C_VEL
LIN {X 0,Y 344.76,Z 566.284,A -85,B 0,C 180,E1 -14147.193,E2 -14147.193} C_VEL
LIN {X 0,Y 343.166,Z 554.873,A -85,B 0,C 180,E1 -14148.335,E2 -14148.335} C_VEL
LIN {X 0,Y 340.133,Z 542.286,A -85,B 0,C 180,E1 -14149.463,E2 -14149.463} C_VEL
LIN {X 0,Y 340.751,Z 536.011,A -85,B 0,C 180,E1 -14153.072,E2 -14153.072} C_VEL
LIN {X 0,Y 341.487,Z 530.818,A -85,B 0,C 180,E1 -14156.263,E2 -14156.263} C_VEL
LIN {X 0,Y 342.307,Z 525.965,A -85,B 0,C 180,E1 -14159.522,E2 -14159.522} C_VEL
LIN {X 0,Y 343.147,Z 521.489,A -85,B 0,C 180,E1 -14162.889,E2 -14162.889} C_VEL
LIN {X 0,Y 343.35,Z 519.041,A -85,B 0,C 180,E1 -14165.04,E2 -14165.04} C_VEL
LIN {X 0,Y 343.051,Z 516.323,A -85,B 0,C 180,E1 -14167.924,E2 -14167.924} C_VEL
LIN {X 0,Y 342.717,Z 514.027,A -85,B 0,C 180,E1 -14171.013,E2 -14171.013} C_VEL
LIN {X 0,Y 342.44,Z 512.295,A -85,B 0,C 180,E1 -14174.251,E2 -14174.251} C_VEL
LIN {X 0,Y 342.207,Z 511.202,A -85,B 0,C 180,E1 -14177.676,E2 -14177.676} C_VEL
LIN {X 0,Y 342.114,Z 510.808,A -85,B 0,C 180,E1 -14181.319,E2 -14181.319} C_VEL
LIN {X 0,Y 342.099,Z 510.927,A -85,B 0,C 180,E1 -14183.433,E2 -14183.433} C_VEL
LIN {X 0,Y 342.012,Z 511.469,A -85,B 0,C 180,E1 -14186.302,E2 -14186.302} C_VEL
LIN {X 0,Y 341.778,Z 512.382,A -85,B 0,C 180,E1 -14189.064,E2 -14189.064} C_VEL
LIN {X 0,Y 341.235,Z 514.274,A -85,B 0,C 180,E1 -14193.057,E2 -14193.057} C_VEL
LIN {X 0,Y 340.743,Z 516.609,A -85,B 0,C 180,E1 -14196.928,E2 -14196.928} C_VEL
LIN {X 0,Y 340.43,Z 519.344,A -85,B 0,C 180,E1 -14200.712,E2 -14200.712} C_VEL
LIN {X 0,Y 340.938,Z 521.138,A -85,B 0,C 180,E1 -14200.879,E2 -14200.879} C_VEL
LIN {X 0,Y 344.543,Z 530.743,A -85,B 0,C 180,E1 -14202.003,E2 -14202.003} C_VEL
LIN {X 0,Y 346.904,Z 539.829,A -85,B 0,C 180,E1 -14203.086,E2 -14203.086} C_VEL
LIN {X 0,Y 347.557,Z 545.006,A -85,B 0,C 180,E1 -14203.706,E2 -14203.706} C_VEL
LIN {X 0,Y 346.316,Z 553.633,A -85,B 0,C 180,E1 -14204.703,E2 -14204.703} C_VEL
LIN {X 0,Y 345.175,Z 561.799,A -85,B 0,C 180,E1 -14205.858,E2 -14205.858} C_VEL
LIN {X 0,Y 343.851,Z 570.153,A -85,B 0,C 180,E1 -14207.307,E2 -14207.307} C_VEL
LIN {X 0,Y 342.721,Z 576.767,A -85,B 0,C 180,E1 -14208.766,E2 -14208.766} C_VEL
LIN {X 0,Y 341.961,Z 581.136,A -85,B 0,C 180,E1 -14209.939,E2 -14209.939} C_VEL
LIN {X 0,Y 341.091,Z 586.27,A -85,B 0,C 180,E1 -14211.707,E2 -14211.707} C_VEL
LIN {X 0,Y 340.397,Z 589.02,A -85,B 0,C 180,E1 -14212.884,E2 -14212.884} C_VEL
LIN {X 0,Y 340.154,Z 591.155,A -85,B 0,C 180,E1 -14214.071,E2 -14214.071} C_VEL
LIN {X 0,Y 340.011,Z 592.669,A -85,B 0,C 180,E1 -14215.257,E2 -14215.257} C_VEL
LIN {X 0,Y 339.701,Z 593.679,A -85,B 0,C 180,E1 -14216.442,E2 -14216.442} C_VEL
LIN {X 0,Y 339.47,Z 594.205,A -85,B 0,C 180,E1 -14217.627,E2 -14217.627} C_VEL
LIN {X 0,Y 339.3,Z 594.258,A -85,B 0,C 180,E1 -14218.813,E2 -14218.813} C_VEL
LIN {X 0,Y 339.231,Z 593.792,A -85,B 0,C 180,E1 -14220,E2 -14220} C_VEL
LIN {X 0,Y 339.192,Z 592.727,A -85,B 0,C 180,E1 -14221.187,E2 -14221.187} C_VEL
LIN {X 0,Y 339.237,Z 590.233,A -85,B 0,C 180,E1 -14222.969,E2 -14222.969} C_VEL
LIN {X 0,Y 339.446,Z 586.354,A -85,B 0,C 180,E1 -14224.751,E2 -14224.751} C_VEL
LIN {X 0,Y 339.551,Z 582.232,A -85,B 0,C 180,E1 -14226.184,E2 -14226.184} C_VEL
LIN {X 0,Y 340.009,Z 576.632,A -85,B 0,C 180,E1 -14227.721,E2 -14227.721} C_VEL
LIN {X 0,Y 340.223,Z 571.332,A -85,B 0,C 180,E1 -14228.913,E2 -14228.913} C_VEL
LIN {X 0,Y 340.667,Z 565.012,A -85,B 0,C 180,E1 -14230.099,E2 -14230.099} C_VEL
LIN {X 0,Y 341.244,Z 556.414,A -85,B 0,C 180,E1 -14231.434,E2 -14231.434} C_VEL
LIN {X 0,Y 341.882,Z 546.768,A -85,B 0,C 180,E1 -14232.616,E2 -14232.616} C_VEL
LIN {X 0,Y 342.448,Z 537.863,A -85,B 0,C 180,E1 -14233.487,E2 -14233.487} C_VEL
LIN {X 0,Y 342.142,Z 532.655,A -85,B 0,C 180,E1 -14233.94,E2 -14233.94} C_VEL
LIN {X 0,Y 340.404,Z 521.81,A -85,B 0,C 180,E1 -14234.703,E2 -14234.703} C_VEL
LIN {X 0,Y 339.404,Z 514.554,A -85,B 0,C 180,E1 -14235.116,E2 -14235.116} C_VEL
LIN {X 0,Y 339.449,Z 510.975,A -85,B 0,C 180,E1 -14238.093,E2 -14238.093} C_VEL
LIN {X 0,Y 339.57,Z 506.539,A -85,B 0,C 180,E1 -14241.873,E2 -14241.873} C_VEL
LIN {X 0,Y 339.786,Z 502.978,A -85,B 0,C 180,E1 -14244.998,E2 -14244.998} C_VEL
LIN {X 0,Y 340.707,Z 506.622,A -85,B 0,C 180,E1 -14246.988,E2 -14246.988} C_VEL
LIN {X 0,Y 340.721,Z 510.449,A -85,B 0,C 180,E1 -14248.995,E2 -14248.995} C_VEL
LIN {X 0,Y 340.485,Z 517.072,A -85,B 0,C 180,E1 -14252.457,E2 -14252.457} C_VEL
LIN {X 0,Y 340.197,Z 524.44,A -85,B 0,C 180,E1 -14256.323,E2 -14256.323} C_VEL
LIN {X 0,Y 340.009,Z 529.488,A -85,B 0,C 180,E1 -14258.892,E2 -14258.892} C_VEL
LIN {X 0,Y 342.15,Z 539.225,A -85,B 0,C 180,E1 -14259.456,E2 -14259.456} C_VEL
LIN {X 0,Y 343.836,Z 548.945,A -85,B 0,C 180,E1 -14260.17,E2 -14260.17} C_VEL
LIN {X 0,Y 344.527,Z 556.65,A -85,B 0,C 180,E1 -14260.847,E2 -14260.847} C_VEL
LIN {X 0,Y 343.597,Z 567.343,A -85,B 0,C 180,E1 -14261.924,E2 -14261.924} C_VEL
LIN {X 0,Y 342.684,Z 576.005,A -85,B 0,C 180,E1 -14263.068,E2 -14263.068} C_VEL
LIN {X 0,Y 342.036,Z 581.943,A -85,B 0,C 180,E1 -14264.014,E2 -14264.014} C_VEL
LIN {X 0,Y 341.341,Z 587.937,A -85,B 0,C 180,E1 -14265.155,E2 -14265.155} C_VEL
LIN {X 0,Y 340.809,Z 592.57,A -85,B 0,C 180,E1 -14266.199,E2 -14266.199} C_VEL
LIN {X 0,Y 340.265,Z 597.66,A -85,B 0,C 180,E1 -14267.607,E2 -14267.607} C_VEL
LIN {X 0,Y 339.942,Z 600.639,A -85,B 0,C 180,E1 -14268.58,E2 -14268.58} C_VEL
LIN {X 0,Y 339.545,Z 604.253,A -85,B 0,C 180,E1 -14270.085,E2 -14270.085} C_VEL
LIN {X 0,Y 339.19,Z 607.384,A -85,B 0,C 180,E1 -14271.939,E2 -14271.939} C_VEL
LIN {X 0,Y 338.905,Z 609.411,A -85,B 0,C 180,E1 -14273.975,E2 -14273.975} C_VEL
LIN {X 0,Y 338.806,Z 609.878,A -85,B 0,C 180,E1 -14276.072,E2 -14276.072} C_VEL
LIN {X 0,Y 338.846,Z 609.428,A -85,B 0,C 180,E1 -14277.366,E2 -14277.366} C_VEL
LIN {X 0,Y 338.944,Z 608.224,A -85,B 0,C 180,E1 -14278.776,E2 -14278.776} C_VEL
LIN {X 0,Y 339.227,Z 605.731,A -85,B 0,C 180,E1 -14280.475,E2 -14280.475} C_VEL
LIN {X 0,Y 339.367,Z 603.631,A -85,B 0,C 180,E1 -14281.555,E2 -14281.555} C_VEL
LIN {X 0,Y 339.769,Z 599.119,A -85,B 0,C 180,E1 -14283.263,E2 -14283.263} C_VEL
LIN {X 0,Y 340.137,Z 594.785,A -85,B 0,C 180,E1 -14284.555,E2 -14284.555} C_VEL
LIN {X 0,Y 340.691,Z 588.944,A -85,B 0,C 180,E1 -14285.957,E2 -14285.957} C_VEL
LIN {X 0,Y 341.26,Z 582.626,A -85,B 0,C 180,E1 -14287.194,E2 -14287.194} C_VEL
LIN {X 0,Y 341.865,Z 575.89,A -85,B 0,C 180,E1 -14288.281,E2 -14288.281} C_VEL
LIN {X 0,Y 342.623,Z 567.147,A -85,B 0,C 180,E1 -14289.434,E2 -14289.434} C_VEL
LIN {X 0,Y 343.369,Z 557.229,A -85,B 0,C 180,E1 -14290.45,E2 -14290.45} C_VEL
LIN {X 0,Y 343.188,Z 552.387,A -85,B 0,C 180,E1 -14290.873,E2 -14290.873} C_VEL
LIN {X 0,Y 341.541,Z 540.514,A -85,B 0,C 180,E1 -14291.75,E2 -14291.75} C_VEL
LIN {X 0,Y 339.774,Z 530.464,A -85,B 0,C 180,E1 -14292.29,E2 -14292.29} C_VEL
LIN {X 0,Y 339.599,Z 529.164,A -85,B 0,C 180,E1 -14292.385,E2 -14292.385} C_VEL
LIN {X 0,Y 339.837,Z 522.004,A -85,B 0,C 180,E1 -14296.406,E2 -14296.406} C_VEL
LIN {X 0,Y 340.018,Z 515.772,A -85,B 0,C 180,E1 -14299.881,E2 -14299.881} C_VEL
LIN {X 0,Y 340.258,Z 509.332,A -85,B 0,C 180,E1 -14303.476,E2 -14303.476} C_VEL
